BEGIN
	//================================================================================
	//SIEMENS AG // (c)Copyright 2019 All Rights Reserved
	//--------------------------------------------------------------------------------
	//Library:       LSimaHydTO
	//Tested with:   S7-15xx
	//Engineering:   TIA Portal  V15
	//Restrictions:  -
	//Requirements:  S7-1500 (FW 2.5)
	//Functionality: - for internal use
	//
	//--------------------------------------------------------------------------------
	//Change log table:
	//
	//Version     Date          Expert in charge    Changes applied
	//01.00.00    24.04.2020    APC_ERLF            First released version
	//================================================================================
	//
	
	#LSimaHydTO_GetSyncAxisCorrection := "LSimaHydTO_GetUnitsCorrection"(lengthUnit:=#axis.Units.LengthUnit,
	                                velocityUnit:=#axis.Units.VelocityUnit,
	                                accelFactor=>#accelFactor);
	
END_FUNCTION

FUNCTION_BLOCK "LSimaHydTO_HydraulicSimulationDrive"
{ S7_Optimized_Access := 'TRUE' }
AUTHOR : APC_ERLF
FAMILY : LSimaHydTO
VERSION : 1.22
   VAR_INPUT 
      enable : Bool;
      initPosition : LReal;
      minPosition : LReal := -1000000000000.0;
      maxPosition : LReal := 1000000000000.0;
      maxVelocity : LReal := 500.0;
      maxForce : LReal := 100.0;
      springDistance : LReal := 1.0;
      externalForce : LReal := 0.0;
      dynamicFrictionFactor : LReal;
      fixedStop : LReal := 1000000000000.0;
      fixedStopInverse : Bool;
      forceInverse : Bool;
      delayTime : LReal;
      cycleTime : UDInt;
      vChar_DB_NUMBER : UInt;
      axisTO : DB_ANY;
   END_VAR

   VAR_OUTPUT 
      busy { ExternalWritable := 'False'} : Bool;
      active { ExternalWritable := 'False'} : Bool;
      error { ExternalWritable := 'False'} : Bool;
      status { ExternalWritable := 'False'} : Word;
      simulatedPosition { ExternalWritable := 'False'} : LReal;
      simulatedForce { ExternalWritable := 'False'} : LReal;
      simulatedVChar { ExternalWritable := 'False'} : UInt;
      forceSensorAnalog_A { ExternalWritable := 'False'} : Word;
      forceSensorAnalog_B { ExternalWritable := 'False'} : Word;
   END_VAR

   VAR_IN_OUT 
      tel2in {InstructionName := 'PD_TEL2_IN'; LibVersion := '4.0'} : PD_TEL2_IN;
      tel2out {InstructionName := 'PD_TEL2_OUT'; LibVersion := '4.0'} : PD_TEL2_OUT;
      tel81in {InstructionName := 'PD_TEL81_IN'; LibVersion := '4.0'} : PD_TEL81_IN;
      tel81out {InstructionName := 'PD_TEL81_OUT'; LibVersion := '4.0'} : PD_TEL81_OUT;
   END_VAR

   VAR 
      statSetPoint { ExternalAccessible := 'False'; ExternalVisible := 'False'; ExternalWritable := 'False'} : LReal;
      statVelSetPoint { ExternalAccessible := 'False'; ExternalVisible := 'False'; ExternalWritable := 'False'} : LReal;
      statActualVChar { ExternalAccessible := 'False'; ExternalVisible := 'False'; ExternalWritable := 'False'} : UInt;
      statSampleTime { ExternalAccessible := 'False'; ExternalVisible := 'False'; ExternalWritable := 'False'} : LReal;
      statActualPosition { ExternalAccessible := 'False'; ExternalVisible := 'False'; ExternalWritable := 'False'} : LReal;
      statActualForce { ExternalAccessible := 'False'; ExternalVisible := 'False'; ExternalWritable := 'False'} : LReal;
      statForceFactor { ExternalAccessible := 'False'; ExternalVisible := 'False'; ExternalWritable := 'False'} : LReal;
      statEnableOld { ExternalAccessible := 'False'; ExternalVisible := 'False'; ExternalWritable := 'False'} : Bool;
      instSetPointPT1 { ExternalAccessible := 'False'; ExternalVisible := 'False'; ExternalWritable := 'False'} : "LSimaHydTO_T1";
      statPosLimitForce { ExternalAccessible := 'False'; ExternalVisible := 'False'; ExternalWritable := 'False'} : LReal;
      statNegLimitForce { ExternalAccessible := 'False'; ExternalVisible := 'False'; ExternalWritable := 'False'} : LReal;
      statFrictionForce { ExternalAccessible := 'False'; ExternalVisible := 'False'; ExternalWritable := 'False'} : LReal;
      instSimpleEncSetValue { ExternalAccessible := 'False'; ExternalVisible := 'False'; ExternalWritable := 'False'} : "LSimaHydTO_SimpleEncTel81";
      statVCharDB { ExternalAccessible := 'False'; ExternalVisible := 'False'; ExternalWritable := 'False'} : DB_ANY;
      statErrorVariant { ExternalAccessible := 'False'; ExternalVisible := 'False'; ExternalWritable := 'False'} : Int;
      instProfiDriveTel2 { ExternalAccessible := 'False'; ExternalVisible := 'False'; ExternalWritable := 'False'} : "LSimaHydTO_ProfiDriveTel2";
      statDriveEnabled { ExternalAccessible := 'False'; ExternalVisible := 'False'; ExternalWritable := 'False'} : Bool;
      statIntVelocityFactor { ExternalAccessible := 'False'; ExternalVisible := 'False'; ExternalWritable := 'False'} : LReal := 1.0;
   END_VAR

   VAR_TEMP 
      tempDeltaPosition : LReal;
      tempMinPos : LReal;
      tempMaxPos : LReal;
      tempActPosOld : LReal;
      tempVCharVar : Variant;
      tempRefToVChar : REF_TO "LSimaHydTO_typeVCharData";
      tempAccFactor : LReal;
   END_VAR

   VAR CONSTANT 
      ERR_INVALID_TYPE_OF_AXIS : Word := 16#8201;
   END_VAR


BEGIN
	//================================================================================
	//SIEMENS AG // (c)Copyright 2019 All Rights Reserved
	//--------------------------------------------------------------------------------
	//Library:       LSimaHydTO
	//Tested with:   S7-15xx
	//Engineering:   TIA Portal  V15
	//Restrictions:  -
	//Requirements:  S7-1500 (FW 2.5)
	//Functionality: Simulation of hydraulic axis   
	//
	//--------------------------------------------------------------------------------
	//Change log table:
	//
	//Version     Date          Expert in charge    Changes applied
	//01.00    15.03.2018    APC_ERLF            First released version
	//01.22    22.04.2020    APC_ERLF            improved: units are taken into account for the control
	//================================================================================
	
	
	IF #enable THEN
	  IF NOT #statEnableOld THEN //positive edge at enable
	    #error := FALSE;
	    #status := 16#0000;
	    #statSampleTime := UDINT_TO_LREAL(#cycleTime) * lreal#1.0E-9;
	    #statActualPosition := #initPosition;
	    
	    CASE TypeOfDB(#axisTO) OF
	            
	        TO_PositioningAxis:
	            #statIntVelocityFactor := "LSimaHydTO_GetPosAxisCorrection"(axis := #axisTO, accelFactor => #tempAccFactor);
	            
	        TO_SynchronousAxis:
	            #statIntVelocityFactor := "LSimaHydTO_GetSyncAxisCorrection"(axis := #axisTO, accelFactor => #tempAccFactor) ;
	            
	        ELSE
	            #error := TRUE;
	            #status := #ERR_INVALID_TYPE_OF_AXIS; // erorr
	            RETURN;
	    END_CASE;
	    
	    #busy := TRUE;
	    #active := TRUE;
	    
	    
	    
	  END_IF;
	  REGION evaluteVChar
	    IF #vChar_DB_NUMBER > 0 THEN
	      #statVCharDB := UINT_TO_DB_ANY(#vChar_DB_NUMBER);
	      #tempVCharVar := DB_ANY_TO_VARIANT(in := #statVCharDB, err => #statErrorVariant);
	      IF #statErrorVariant = 0 THEN
	        #tempRefToVChar ?= #tempVCharVar;
	        
	        IF TypeOf(#tempVCharVar) <> LSimaHydTO_typeVCharData THEN
	          #statErrorVariant := 8200;
	        END_IF;
	      END_IF;
	      IF #statErrorVariant <> 0 THEN
	        #statActualVChar := 0;
	        
	      ELSE
	        // check consinsesty of VChar
	        IF #tempRefToVChar^.MaxIdx < 1 OR #tempRefToVChar^.VelocityLimitPositive <= #tempRefToVChar^.VelocityLimitNegative THEN
	          #statActualVChar := 0;
	        ELSE
	          #statActualVChar := #vChar_DB_NUMBER;
	        END_IF;
	      END_IF;
	    ELSE
	      #statActualVChar := 0;
	    END_IF;
	    
	    #instProfiDriveTel2(setpoint => #statSetPoint,
	                        driveEnabled => #statDriveEnabled,
	                        tel2in := #tel2in,
	                        tel2out := #tel2out);
	    
	    
	    
	    IF #statActualVChar = 0 THEN
	      #statVelSetPoint := "LSimaHydTO_Scale"(input := #statSetPoint,
	                                           inBegin := -100.0,
	                                           inEnd := 100.0,
	                                           valBegin := - #maxVelocity,
	                                           valEnd := #maxVelocity);
	    ELSE
	      
	      #statVelSetPoint := "LSimaHydTO_VcharInverse"(qOutput := #statSetPoint, VChar := #tempRefToVChar^);
	      #statVelSetPoint := LIMIT(MN := - #maxVelocity, IN := #statVelSetPoint, MX := #maxVelocity);
	    END_IF;
	    #statVelSetPoint := #statVelSetPoint / #statIntVelocityFactor;
	    #simulatedVChar := #statActualVChar;
	  END_REGION
	  
	  #statActualForce := LIMIT(MN := - #maxForce, IN := #statActualForce, MX := #maxForce);
	  IF (#statActualForce > 0.0 AND
	    #statVelSetPoint > 0.0)
	    OR
	    (#statActualForce < 0.0 AND
	    #statVelSetPoint < 0.0)
	  THEN
	    #statForceFactor := MAX(IN1 := 0.0, IN2 := SQRT((#maxForce - ABS(#statActualForce)) / #maxForce));
	  ELSE
	    #statForceFactor := 1.0;
	  END_IF;
	  
	  
	  #instSetPointPT1(enable := #enable AND #delayTime > 0.0,
	                   inputValue := #statVelSetPoint,
	                   timeConstant := #delayTime,
	                   sampleTime := #statSampleTime
	                   // ,outputValue => 
	                   // ,active => 
	                   // ,error => 
	                   );
	  
	  #tempDeltaPosition := (#instSetPointPT1.outputValue) * #statSampleTime * #statForceFactor;
	  
	  //calculate AND LIMIT actual postition
	  #tempActPosOld := #statActualPosition;
	  
	  IF #fixedStopInverse THEN
	    #tempMinPos := LIMIT(MN := #minPosition
	                         , IN := #fixedStop
	                         , MX := #maxPosition);
	    #tempMaxPos := #maxPosition;
	  ELSE
	    #tempMinPos := #minPosition;
	    #tempMaxPos := LIMIT(MN := #minPosition
	                         , IN := #fixedStop
	                         , MX := #maxPosition);
	    
	  END_IF;
	  #statActualPosition := LIMIT( MN := #tempMinPos
	                              , IN := #tempActPosOld + #tempDeltaPosition
	                              , MX := #tempMaxPos
	                              );
	  #statFrictionForce := #dynamicFrictionFactor*(#statActualPosition - #tempActPosOld)/#statSampleTime;
	  IF #maxForce > 0.0
	    AND #springDistance > 0.0
	  THEN
	    
	    IF (#tempMaxPos - #statActualPosition) < #springDistance THEN
	      
	      #statPosLimitForce := LIMIT(MN := 0.0
	                                  , IN := (1 - (#tempMaxPos - #statActualPosition) / #springDistance) * #maxForce
	                                  , MX := #maxForce);
	    ELSE
	      #statPosLimitForce := 0.0;
	    END_IF;
	    IF (#statActualPosition - #tempMinPos) < #springDistance THEN
	      #statNegLimitForce := -LIMIT(MN := 0.0
	                                  , IN :=  (1 - (#statActualPosition - #tempMinPos) / #springDistance) * #maxForce
	                                  , MX := #maxForce);
	    ELSE
	      #statNegLimitForce := 0.0;
	    END_IF;
	    
	    #statActualForce := #externalForce + #statNegLimitForce + #statPosLimitForce + #statFrictionForce;
	    
	  ELSE
	    #statActualForce := #externalForce + #statFrictionForce;
	  END_IF;
	  
	  IF #forceInverse THEN
	    #statActualForce := -1.0 * #statActualForce;
	  END_IF;
	  //write actual position to technology object
	  
	  #simulatedPosition := #statActualPosition;
	  #simulatedForce := LIMIT(MN := - #maxForce, IN := #statActualForce, MX := #maxForce);
	  
	  IF #maxForce > 0.0 THEN
	    IF #simulatedForce >= 0.0 THEN
	      #forceSensorAnalog_A := INT_TO_WORD(LREAL_TO_INT(#simulatedForce * 27648.0 / #maxForce));
	      #forceSensorAnalog_B := 0;
	    ELSE
	      #forceSensorAnalog_B := INT_TO_WORD(LREAL_TO_INT(ABS(#simulatedForce) * 27648.0 / #maxForce));
	      #forceSensorAnalog_A := 0;
	    END_IF;
	  ELSE
	    #forceSensorAnalog_A := 0;
	    #forceSensorAnalog_B := 0;
	  END_IF;
	  
	  #instSimpleEncSetValue(position := #simulatedPosition,
	                         init := #enable AND NOT #statEnableOld,
	                         axis:=#axisTO,
	                         status=>#status,
	                         tel81in := #tel81in,
	                         tel81out := #tel81out);
	  
	  
	  
	ELSE
	  IF #statEnableOld THEN //negative edge
	    #busy := FALSE;
	    #active := FALSE;
	    #simulatedVChar := 0;
	    
	    #statActualPosition := 0.0;
	    #statActualForce := 0.0;
	    #simulatedPosition := 0.0;
	    #simulatedForce := 0.0;
	    #forceSensorAnalog_A := 0;
	    #forceSensorAnalog_B := 0;
	  END_IF;
	END_IF;
	
	
	#statEnableOld := #enable;
	
	
	
	
	
	
END_FUNCTION_BLOCK

FUNCTION_BLOCK "LSimaHydTO_ProfiDriveTel2"
{ S7_Optimized_Access := 'FALSE' }
AUTHOR : APC_ERLF
FAMILY : LSimaHydTO
VERSION : 1.0
   VAR_OUTPUT 
      setpoint { ExternalAccessible := 'False'; ExternalVisible := 'False'; ExternalWritable := 'False'} : LReal;
      driveEnabled { ExternalAccessible := 'False'; ExternalVisible := 'False'; ExternalWritable := 'False'} : Bool;
   END_VAR

   VAR_IN_OUT 
      tel2in {InstructionName := 'PD_TEL2_IN'; LibVersion := '4.0'} : PD_TEL2_IN;
      tel2out {InstructionName := 'PD_TEL2_OUT'; LibVersion := '4.0'} : PD_TEL2_OUT;
   END_VAR

   VAR 
      statZSW1 {InstructionName := 'PD_ZSW1'; LibVersion := '4.0'; ExternalAccessible := 'False'; ExternalVisible := 'False'; ExternalWritable := 'False'} : PD_ZSW1;
      statWZSW1 { ExternalAccessible := 'False'; ExternalVisible := 'False'; ExternalWritable := 'False'} AT statZSW1 : Word;
   END_VAR

   VAR_TEMP 
      tempNsollSigned : DInt;
   END_VAR

   VAR CONSTANT 
      ZSW1_S1 : Word := 2#0000_0011_0111_0000;
      ZSW1_S2 : Word := 2#0000_0011_0011_0001;
      ZSW1_S3 : Word := 2#0000_0011_0011_0011;
      ZSW1_S4 : Word := 2#0000_0011_0011_0111;
      C_100_PROZENT : LReal := 10737418.24;
   END_VAR


BEGIN
	//================================================================================
	//SIEMENS AG // (c)Copyright 2019 All Rights Reserved
	//--------------------------------------------------------------------------------
	//Library:       LSimaHydTO
	//Tested with:   S7-15xx
	//Engineering:   TIA Portal  V15
	//Restrictions:  -
	//Requirements:  S7-1500 (FW 2.5)
	//Functionality: Support of drive transmitter   
	//
	//--------------------------------------------------------------------------------
	//Change log table:
	//
	//Version     Date          Expert in charge    Changes applied
	//01.00.00    29.03.2017    APC_ERLF            First released version
	//================================================================================
	
	
	IF #tel2out.STW1.NoCoastStop AND #tel2out.STW1.NoQuickStop THEN
	    IF #tel2out.STW1.On THEN
	        IF #tel2out.STW1.EnableOperation THEN
	            #statWZSW1 := #ZSW1_S4;             // operation
	            #driveEnabled := TRUE;
	        ELSE
	            #statWZSW1 := #ZSW1_S3;             // switched on
	        END_IF;
	    ELSE
	        #statWZSW1 := #ZSW1_S2;                 // ready for switch on
	    END_IF;
	ELSE
	    #statWZSW1 := #ZSW1_S1;                 // coast stop, quick stop
	    #driveEnabled := FALSE;
	END_IF;
	#tel2in.ZSW1 := #statZSW1;
	//-----------------  Interface -----------  
	#tempNsollSigned := DWORD_TO_DINT(#tel2out.NSOLL_B); // NSOLL is really a signed DINT
	#setpoint := DINT_TO_LREAL(#tempNsollSigned)/#C_100_PROZENT;      // desired speed 
	IF #statWZSW1 = #ZSW1_S4 THEN
	  #tel2in.NIST_B := #tel2out.NSOLL_B;
	ELSE
	  #tel2in.NIST_B := 0;
	END_IF;
	
	
END_FUNCTION_BLOCK

FUNCTION "Scale" : Void   // FC1, LAD
{ S7_Optimized_Access := 'TRUE' }
VERSION : 0.1
// stored: AutoNumber true, IsIECCheckEnabled false, SetENOAutomatically false, UDAEnableTagReadback false
   VAR_OUTPUT
      Scale_Out : Real;
   END_VAR
   VAR_TEMP
      AUX : Real;
   END_VAR
BEGIN

REGION Network 1
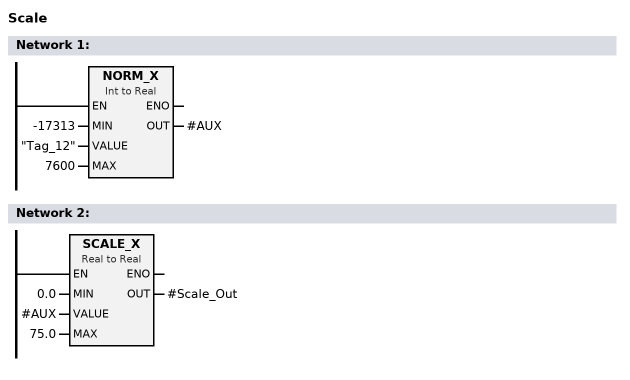
   RUNG wire#powerrail
      { S7_Templates := "[SrcType := Int, DestType := Real]" } Normalize(min := -17313, value := "Tag_12", max := 7600, out => #AUX)
   END_RUNG
   // the same network as SCL:
   #AUX := NORM_X(MIN := -17313, VALUE := "Tag_12", MAX := 7600);
END_REGION

REGION Network 2
   RUNG wire#powerrail
      { S7_Templates := "[SrcType := Real, DestType := Real]" } Scale(min := 0.0, value := #AUX, max := 75.0, out => #Scale_Out)
   END_RUNG
   // the same network as SCL:
   #Scale_Out := SCALE_X(MIN := 0.0, VALUE := #AUX, MAX := 75.0);
END_REGION
END_FUNCTION

ORGANIZATION_BLOCK "SimaHydTO_Main_HMI"   // OB124, LAD, ProgramCycle
TITLE = SimaHydTO_Main_HMI
{ S7_Optimized_Access := 'TRUE' }
FAMILY : SimaHydTO
VERSION : 1.0
// Organization block information: See Organization block network 1
// stored: AutoNumber true, IsIECCheckEnabled false, SetENOAutomatically false
   VAR_INPUT
      Initial_Call : Bool;   // Initial call of this OB
      Remanence : Bool;   // =True, if remanent data are available
   END_VAR
BEGIN

REGION Network 1 (SCL): SimaHydTO - HMI Interface
   //=============================================================================
   //SIEMENS AG
   //(c)Copyright 2016 All Rights Reserved
   //-----------------------------------------------------------------------------
   //Library:       OB of LSimaHydTO_HMI
   //Tested with:   S7-1500 V2.5
   //Engineering:   TIA Portal V15
   //Restrictions:  -
   //Requirements:  S7-1500(T)
   //Functionality: Connection between HMI and PLC program
   //-----------------------------------------------------------------------------
   //Change log table:
   //Version  Date       Expert in charge Changes applied
   //01.00.00 18.07.2019 ArSc             First released version
   //=============================================================================
END_REGION

REGION Network 2: SimaHydTO - HMI Interface: Function calls of HMI functionality
   // Controlling the functionality of SimaHydTO via HMI
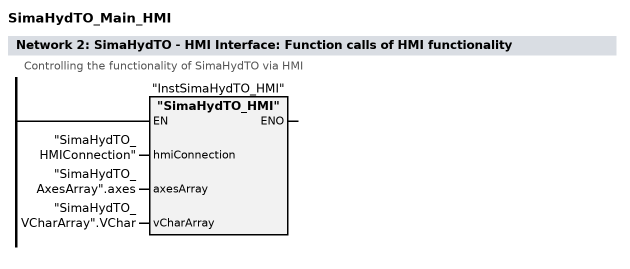
   RUNG wire#powerrail
      "InstSimaHydTO_HMI"(hmiConnection := "SimaHydTO_HMIConnection", axesArray := "SimaHydTO_AxesArray".axes, vCharArray := "SimaHydTO_VCharArray".VChar)
   END_RUNG
   // the same network as SCL:
   "InstSimaHydTO_HMI"(hmiConnection := "SimaHydTO_HMIConnection",   // "SimaHydTO_HMI"
                       axesArray := "SimaHydTO_AxesArray".axes,
                       vCharArray := "SimaHydTO_VCharArray".VChar);
END_REGION
END_ORGANIZATION_BLOCK

FUNCTION_BLOCK "SimaHydTO_HMI"
{ S7_Optimized_Access := 'TRUE' }
FAMILY : SimaHydTO
VERSION : 1.0
   VAR_IN_OUT 
      hmiConnection : "SimaHydTO_typeHMIConnection";
      axesArray : Array[*] of "SimaHydTO_typeAxesArray";
      vCharArray : Array[*] of "SimaHydTO_typeVCharArray";
   END_VAR

   VAR 
      statInitObjects { ExternalAccessible := 'False'; ExternalVisible := 'False'; ExternalWritable := 'False'} : Bool := TRUE;
      instHmiAxisSelector { ExternalAccessible := 'False'; ExternalVisible := 'False'; ExternalWritable := 'False'} : "SimaHydTO_HmiAxisSelector";
      instHmiVCharSelector { ExternalAccessible := 'False'; ExternalVisible := 'False'; ExternalWritable := 'False'} : "SimaHydTO_HmiVCharSelector";
      instBasicAxisControl { ExternalAccessible := 'False'; ExternalVisible := 'False'; ExternalWritable := 'False'} : "SimaHydTO_BasicAxisControl";
      instVCharMeasurement { ExternalAccessible := 'False'; ExternalVisible := 'False'; ExternalWritable := 'False'} : "SimaHydTO_VCharMeasurement";
      instVCharEditor { ExternalAccessible := 'False'; ExternalVisible := 'False'; ExternalWritable := 'False'} : "SimaHydTO_VCharEditor";
      instAdvancedAxisControl { ExternalAccessible := 'False'; ExternalVisible := 'False'; ExternalWritable := 'False'} : "SimaHydTO_AdvancedAxisControl";
      instParameterSettings { ExternalAccessible := 'False'; ExternalVisible := 'False'; ExternalWritable := 'False'} : "SimaHydTO_ParameterSettings";
      instFindVChars { ExternalAccessible := 'False'; ExternalVisible := 'False'; ExternalWritable := 'False'} : "SimaHydTO_FindObjects";
      instVCharManagement { ExternalAccessible := 'False'; ExternalVisible := 'False'; ExternalWritable := 'False'} : "SimaHydTO_VCharManagement";
   END_VAR

   VAR_TEMP 
      tempVariant : Variant;
      tempErrorVariant : Int;
      tempDbAny : DB_ANY;
      tempHydAxisData : REF_TO "LSimaHydTO_typeAxisData";
   END_VAR


BEGIN
	//=============================================================================
	//SIEMENS AG
	//(c)Copyright 2016 All Rights Reserved
	//-----------------------------------------------------------------------------
	//Library:       SimaHydTO_HMI
	//Tested with:   S7-1500 V2.5
	//Engineering:   TIA Portal V15
	//Restrictions:  -
	//Requirements:  S7-1500(T)
	//Functionality: Connection between HMI and PLC program
	//-----------------------------------------------------------------------------
	//Change log table:
	//Version  Date       Expert in charge Changes applied
	//01.00.00 12.07.2019 ArSc             First released version
	//=============================================================================
	
	#instFindVChars(execute := #statInitObjects,
	                axesArray := #axesArray,
	                vCharArray := #vCharArray);
	IF NOT #instFindVChars.busy THEN
	  #statInitObjects := FALSE;
	END_IF;
	
	//=============================================================================
	//Axis selector
	//=============================================================================
	
	//Axis selection 
	#instHmiAxisSelector(selector := #hmiConnection.AxisSelector,
	                     axesArray := #axesArray);
	
	
	
	//===================================================================================
	//evalute objects
	//
	
	#tempDbAny := #hmiConnection.AxisSelector.Status.selectedAxis;
	#tempVariant := DB_ANY_TO_VARIANT(in := #tempDbAny, err => #tempErrorVariant);
	
	IF TypeOf(#tempVariant) = LSimaHydTO_typeAxisData THEN
	  #tempHydAxisData ?= #tempVariant;
	  
	END_IF;
	//=============================================================================
	//Basic axis control
	//=============================================================================
	
	//Check axis selection
	IF (#hmiConnection.AxisSelector.Status.dataValid = True)
	THEN
	  IF (#hmiConnection.AxisSelector.Status.selectionChanged = True)
	  THEN
	    CASE #hmiConnection.AxisSelector.Status.selectedTypeOfAxis OF
	      2: //posaxis
	        #hmiConnection.AxisToData.axisUnits := "SimaHydTO_GetAxisToUnits_PosAxis"(#hmiConnection.AxisSelector.Status.selectedTO_Axis);
	        
	      3: // syncaxis
	        #hmiConnection.AxisToData.axisUnits := "SimaHydTO_GetAxisToUnits_SyncAxis"(#hmiConnection.AxisSelector.Status.selectedTO_Axis);
	        
	    END_CASE;
	    #hmiConnection.AxisToData.typeOfAxis := #hmiConnection.AxisSelector.Status.selectedTypeOfAxis;
	  END_IF;
	  
	  // Axis animation
	    "SimaHydTO_HmiAxisAnimation"(hmiConnection := #hmiConnection,
	                                 axisData := #tempHydAxisData^);
	    
	  
	  
	  //Transfer data between axis and HMI
	  #instBasicAxisControl(hmiConnection := #hmiConnection,
	                        axisData := #tempHydAxisData^,
	                        axesArray := #axesArray);
	  
	  
	  
	  //=============================================================================
	  //VChar measurement
	  //=============================================================================
	  
	  //Call function block
	  #instVCharMeasurement(hmiConnection := #hmiConnection,
	                        axisData := #tempHydAxisData^,
	                        axesArray:=#axesArray,
	                        vCharArray := #vCharArray);
	  
	  
	  
	  //=============================================================================
	  //Advanced axis control
	  //=============================================================================
	  #instAdvancedAxisControl(hmiConnection := #hmiConnection,
	                           axisData := #tempHydAxisData^,
	                           axesArray := #axesArray);
	  
	  
	  #instVCharManagement(hmiConnection:=#hmiConnection,
	                       axisData:=#tempHydAxisData^,
	                       vCharArray:=#vCharArray);
	
	  
	ELSE
	  //In case of no valid data of axis selection, do nothing...
	  ;
	END_IF;
	
	//=============================================================================
	//VChar editor
	//=============================================================================
	
	//Do function...
	#instVCharEditor(hmiConnection := #hmiConnection,
	                 vCharArray := #vCharArray);
	
	
	
	//=============================================================================
	//Parameter settings
	//=============================================================================
	
	//Check axis selection
	//Do function...
	#instParameterSettings(hmiConnection := #hmiConnection,
	                       axisData := #tempHydAxisData^,
	                       VCharArray := #vCharArray);
	
	
	
	
	
END_FUNCTION_BLOCK

FUNCTION_BLOCK "SimaHydTO_HmiAxisSelector"
{ S7_Optimized_Access := 'TRUE' }
FAMILY : SimaHydTO
VERSION : 1.0
   VAR_IN_OUT 
      selector : "SimaHydTO_typeHMIConnectionAxisSelector";
      axesArray : Array[*] of "SimaHydTO_typeAxesArray";
   END_VAR

   VAR 
      statFirstRunDone { ExternalAccessible := 'False'; ExternalVisible := 'False'; ExternalWritable := 'False'} : Bool;
      statActualAxisIndex { ExternalAccessible := 'False'; ExternalVisible := 'False'; ExternalWritable := 'False'} : Int;
      statArrayMinIndex { ExternalAccessible := 'False'; ExternalVisible := 'False'; ExternalWritable := 'False'} : Int;
      statArrayMaxIndex { ExternalAccessible := 'False'; ExternalVisible := 'False'; ExternalWritable := 'False'} : Int;
      statPreviousObjectOld { ExternalAccessible := 'False'; ExternalVisible := 'False'; ExternalWritable := 'False'} : Bool;
      statNextObjectOld { ExternalAccessible := 'False'; ExternalVisible := 'False'; ExternalWritable := 'False'} : Bool;
      statExecuteDirectIndexSelectionOld { ExternalAccessible := 'False'; ExternalVisible := 'False'; ExternalWritable := 'False'} : Bool;
      statActualAxisIndexOld { ExternalAccessible := 'False'; ExternalVisible := 'False'; ExternalWritable := 'False'} : Int;
   END_VAR

   VAR_TEMP 
      tempVariant : Variant;
      tempErrorVariant : Int;
      tempDbAny : DB_ANY;
      tempHydAxisData : REF_TO "LSimaHydTO_typeAxisData";
   END_VAR

   VAR CONSTANT 
      ERROR_AXIS_INDEX : Int := 0;
      ERROR_SELECTED_HYDAXIS : DB_ANY := 0;
      ERROR_SELECTED_HYDAXIS_INTEGER : UInt := 0;
      ERROR_SELECTED_HYDAXIS_NAME : WString := WSTRING#'';
      ERROR_SELECTED_AXISTO : DB_ANY := 0;
      ERROR_SELECTED_AXISTO_INTEGER : UInt := 0;
      ERROR_SELECTED_AXISTO_TYPE : Int := 0;
      ERROR_SELECTED_VCHAR : DB_ANY := 0;
      ERROR_SELECTED_VCHAR_INTEGER : UInt := 0;
   END_VAR


BEGIN
	//=============================================================================
	//SIEMENS AG
	//(c)Copyright 2016 All Rights Reserved
	//-----------------------------------------------------------------------------
	//Library:       SimaHydTO_HMI
	//Tested with:   S7-1500 V2.5
	//Engineering:   TIA Portal V15
	//Restrictions:  -
	//Requirements:  S7-1500(T)
	//Functionality: Selection of hydraulic axis out of axis array
	//-----------------------------------------------------------------------------
	//Change log table:
	//Version  Date       Expert in charge Changes applied
	//01.00.00 12.07.2019 ArSc             First released version
	//=============================================================================
	
	
	//Array detection and initialization
	IF (#statFirstRunDone = False)
	THEN
	  //Get MIN and MAX of array indices
	  #statArrayMinIndex := DINT_TO_INT(LOWER_BOUND(ARR := #axesArray, DIM := 1));
	  #statArrayMaxIndex := DINT_TO_INT(UPPER_BOUND(ARR := #axesArray, DIM := 1));
	  //Set default value of actual axis index
	  #statActualAxisIndex := #statArrayMinIndex;
	  #statActualAxisIndexOld := #statArrayMinIndex-1;
	  //Mark first run of function block
	  #statFirstRunDone := True;
	  #selector.Status.dataError := False;
	  #selector.Status.dataValid := False;
	END_IF;
	  //Select axis (in axis data array)
	  //Previous axis
	IF ((#selector.Command.previousObject = True)
	    AND (#statPreviousObjectOld = False)
	    AND (#selector.Command.nextObject = False)
	    AND (#selector.Command.executeDirectIndexSelection = False))
	  THEN
	    //Decrement actual axis index
	    #statActualAxisIndex := #statActualAxisIndex - INT#1;
	    //Check index minimum
	    IF (#statActualAxisIndex < #statArrayMinIndex)
	    THEN
	      //Select last axis by index
	      #statActualAxisIndex := #statArrayMaxIndex;
	    END_IF;
	    //Next axis  
	  ELSIF ((#selector.Command.nextObject = True)
	    AND (#statNextObjectOld = False)
	    AND (#selector.Command.previousObject = False)
	    AND (#selector.Command.executeDirectIndexSelection = False))
	  THEN
	    //Increment actual axis index
	    #statActualAxisIndex := #statActualAxisIndex + INT#1;
	    //Check index minimum
	    IF (#statActualAxisIndex > #statArrayMaxIndex)
	    THEN
	      //Select first axis by index
	      #statActualAxisIndex := #statArrayMinIndex;
	    END_IF;
	    //Direct selection
	  ELSIF ((#selector.Command.executeDirectIndexSelection = True)
	    AND (#statExecuteDirectIndexSelectionOld = False)
	    AND (#selector.Command.nextObject = False)
	    AND (#selector.Command.previousObject = False))
	  THEN
	    IF ((#selector.Command.directIndexSelection >= #statArrayMinIndex)
	      AND (#selector.Command.directIndexSelection <= #statArrayMaxIndex))
	    THEN
	      //Set axis index directly
	      #statActualAxisIndex := #selector.Command.directIndexSelection;
	    END_IF;
	  END_IF;
	
	  #selector.Status.selectionChanged := FALSE;
	  IF #statActualAxisIndex <> #statActualAxisIndexOld
	    AND #axesArray[#statActualAxisIndex].initialized
	  THEN
	    //Write function block output
	    #selector.Status.actualAxisIndex := #statActualAxisIndex;
	    #tempDbAny := #axesArray[#statActualAxisIndex].axisData;
	    
	    #selector.Status.selectedAxis := #tempDbAny;
	    #selector.Status.selectedAxisInteger := DB_ANY_TO_UINT(#tempDbAny);
	    
	    //Get axis data
	    #tempVariant := DB_ANY_TO_VARIANT(in := #tempDbAny, err => #tempErrorVariant);
	    
	    IF TypeOf(#tempVariant) = LSimaHydTO_typeAxisData THEN
	      #tempHydAxisData ?= #tempVariant;
	      
	      //Read hydraulic axis name
	      #selector.Status.selectedAxisName := #tempHydAxisData^.Name;
	      //Read connected technology object axis
	      
	      CASE TypeOfDB(#tempHydAxisData^.TO_Axis) OF
	          
	        TO_PositioningAxis:
	          #selector.Status.selectedTO_Axis := #tempHydAxisData^.TO_Axis;
	          #selector.Status.selectedAxisTOInteger := DB_ANY_TO_UINT(#selector.Status.selectedTO_Axis);
	          #selector.Status.selectedTypeOfAxis := 2;
	          
	          #selector.Status.dataValid := TRUE;
	          
	        TO_SynchronousAxis:
	          #selector.Status.selectedTO_Axis := #tempHydAxisData^.TO_Axis;
	          #selector.Status.selectedAxisTOInteger := DB_ANY_TO_UINT(#selector.Status.selectedTO_Axis);
	          #selector.Status.selectedTypeOfAxis := 3;
	          #selector.Status.dataValid := TRUE;
	          
	        ELSE
	          #selector.Status.selectedTO_Axis := 0;
	          #selector.Status.selectedAxisTOInteger := 0;
	          #selector.Status.selectedTypeOfAxis := 0;
	          #selector.Status.dataValid := FALSE;
	          
	      END_CASE;
	      //Read active valve characteristics
	      #selector.Status.selectedVChar := #tempHydAxisData^.ValveCharacteristic.DB_NUMBER;
	      #selector.Status.selectedVCharInteger := DB_ANY_TO_UINT(#selector.Status.selectedVChar);
	      
	      //Write function block output
	      #selector.Status.dataError := False;
	  //    #selector.Status.dataValid := TRUE;
	      #selector.Status.selectionChanged := TRUE;
	    ELSE
	      //error handling
	      #selector.Status.dataError := True;
	      #selector.Status.dataValid := False;
	      
	      #selector.Status.actualAxisIndex := #statActualAxisIndex;
	      #selector.Status.selectedAxis := #ERROR_SELECTED_HYDAXIS;
	      #selector.Status.selectedAxisInteger := #ERROR_SELECTED_HYDAXIS_INTEGER;
	      #selector.Status.selectedAxisName := #ERROR_SELECTED_HYDAXIS_NAME;
	      #selector.Status.selectedTO_Axis := #ERROR_SELECTED_AXISTO;
	      #selector.Status.selectedAxisTOInteger := #ERROR_SELECTED_AXISTO_INTEGER;
	      #selector.Status.selectedTypeOfAxis := #ERROR_SELECTED_AXISTO_TYPE;
	      #selector.Status.selectedVChar := #ERROR_SELECTED_VCHAR;
	      #selector.Status.selectedVCharInteger := #ERROR_SELECTED_VCHAR_INTEGER;
	      
	    END_IF;
	    //Save AxisIndex for edge control
	    #statActualAxisIndexOld := #statActualAxisIndex;
	    
	  END_IF;
	
	
	//-----------------------------------------------------------------------------
	//Function block system functions
	//-----------------------------------------------------------------------------
	
	//Save signals for edge control
	  #statPreviousObjectOld := #selector.Command.previousObject;
	  #statNextObjectOld := #selector.Command.nextObject;
	  #statExecuteDirectIndexSelectionOld := #selector.Command.executeDirectIndexSelection;
	
	
	
END_FUNCTION_BLOCK

FUNCTION_BLOCK "SimaHydTO_HmiVCharSelector"
{ S7_Optimized_Access := 'TRUE' }
FAMILY : SimaHydTO
VERSION : 1.0
   VAR_INPUT 
      command { ExternalAccessible := 'False'; ExternalVisible := 'False'; ExternalWritable := 'False'} : "SimaHydTO_typeHMIConnectionVCharSelectorCommand";
   END_VAR

   VAR_IN_OUT 
      status : "SimaHydTO_typeHMIConnectionVCharSelectorStatus";
      vCharArray : Array[*] of "SimaHydTO_typeVCharArray";
   END_VAR

   VAR 
      statFirstRunDone { ExternalAccessible := 'False'; ExternalVisible := 'False'; ExternalWritable := 'False'} : Bool;
      statActualVCharIndex { ExternalAccessible := 'False'; ExternalVisible := 'False'; ExternalWritable := 'False'} : Int;
      statArrayMinIndex { ExternalAccessible := 'False'; ExternalVisible := 'False'; ExternalWritable := 'False'} : Int;
      statArrayMaxIndex { ExternalAccessible := 'False'; ExternalVisible := 'False'; ExternalWritable := 'False'} : Int;
      statPreviousObjectOld { ExternalAccessible := 'False'; ExternalVisible := 'False'; ExternalWritable := 'False'} : Bool;
      statNextObjectOld { ExternalAccessible := 'False'; ExternalVisible := 'False'; ExternalWritable := 'False'} : Bool;
      statExecuteDirectIndexSelectionOld { ExternalAccessible := 'False'; ExternalVisible := 'False'; ExternalWritable := 'False'} : Bool;
   END_VAR

   VAR_TEMP 
      tempVariant : Variant;
      tempErrorVariant : Int;
      tempDbAny : DB_ANY;
      tempVCharData : REF_TO "LSimaHydTO_typeVCharData";
      tempIndexChanged : Bool;
   END_VAR

   VAR CONSTANT 
      ERROR_VCHAR_INDEX : Int := 0;
      ERROR_SELECTED_VCHAR : DB_ANY := 0;
      ERROR_SELECTED_VCHAR_INTEGER : UInt := 0;
      ERROR_SELECTED_VCHAR_NAME : WString := WSTRING#'';
   END_VAR


BEGIN
	//=============================================================================
	//SIEMENS AG
	//(c)Copyright 2016 All Rights Reserved
	//-----------------------------------------------------------------------------
	//Library:       SimaHydTO_HMI
	//Tested with:   S7-1500 V2.5
	//Engineering:   TIA Portal V15
	//Restrictions:  -
	//Requirements:  S7-1500(T)
	//Functionality: Selection of VChar (valve characteristics) controlled via HMI
	//-----------------------------------------------------------------------------
	//Change log table:
	//Version  Date       Expert in charge Changes applied
	//01.00.00 12.07.2019 ArSc             First released version
	//=============================================================================
	
	
	//Array detection and initialization
	IF (#statFirstRunDone = False)
	THEN
	  //Get MIN and MAX of array indices
	  #statArrayMinIndex := DINT_TO_INT(LOWER_BOUND(ARR := #vCharArray, DIM := 1));
	  #statArrayMaxIndex := DINT_TO_INT(UPPER_BOUND(ARR := #vCharArray, DIM := 1));
	  //Set default value of actual axis index
	  #statActualVCharIndex := #statArrayMinIndex;
	  //Mark first run of function block
	  IF #vCharArray[#statActualVCharIndex].initialized THEN
	    #statFirstRunDone := True;
	    #tempIndexChanged := TRUE;
	  END_IF;
	  
	ELSE
	  //Select axis (in axis data array)
	  //Previous axis
	  IF (#command.previousObject
	    AND  NOT #statPreviousObjectOld)
	  THEN
	    //Decrement actual axis index
	    #statActualVCharIndex := #statActualVCharIndex - INT#1;
	    //Check index minimum
	    IF (#statActualVCharIndex < #statArrayMinIndex)
	    THEN
	      //Select last axis by index
	      #statActualVCharIndex := #statArrayMaxIndex;
	    END_IF;
	    #tempIndexChanged := TRUE;
	  //Next axis  
	  ELSIF (#command.nextObject
	    AND NOT #statNextObjectOld)
	  THEN
	    //Increment actual axis index
	    #statActualVCharIndex := #statActualVCharIndex + INT#1;
	    //Check index minimum
	    IF (#statActualVCharIndex > #statArrayMaxIndex)
	    THEN
	      //Select first axis by index
	      #statActualVCharIndex := #statArrayMinIndex;
	    END_IF;
	    #tempIndexChanged := TRUE;
	  //Direct selection
	  ELSIF (#command.executeDirectIndexSelection
	    AND NOT #statExecuteDirectIndexSelectionOld)
	  THEN
	    IF ((#command.directIndexSelection >= #statArrayMinIndex)
	      AND (#command.directIndexSelection <= #statArrayMaxIndex))
	    THEN
	      //Set axis index directly
	      #statActualVCharIndex := DINT_TO_INT(#command.directIndexSelection);
	      #tempIndexChanged := TRUE;
	    END_IF;
	  END_IF;
	END_IF;
	
	
	IF (#statFirstRunDone)
	THEN
	  //Write function block output
	  #status.actualVCharIndex := #statActualVCharIndex;
	  IF #tempIndexChanged  THEN
	    //Get VChar data
	    #tempDbAny := #vCharArray[#status.actualVCharIndex].VChar_DB;
	    #tempVariant := DB_ANY_TO_VARIANT(in := #tempDbAny, err => #tempErrorVariant);
	    
	    IF TypeOf(#tempVariant) = LSimaHydTO_typeVCharData THEN
	      #tempVCharData ?= #tempVariant;
	      
	      #status.selectedVChar := #vCharArray[#status.actualVCharIndex].VChar_DB;
	      #status.selectedVCharName := #tempVCharData^.Name;
	      #status.selectedVCharInteger := DB_ANY_TO_UINT(#status.selectedVChar);
	      
	      //Write function block output
	      #status.dataError := False;
	      #status.dataValid := True;
	      
	    ELSE
	      //error handling
	      #status.dataError := True;
	      #status.dataValid := False;
	      
	      // #actualVCharIndex := #ERROR_VCHAR_INDEX;
	      #status.selectedVChar := #ERROR_SELECTED_VCHAR;
	      #status.selectedVCharInteger := #ERROR_SELECTED_VCHAR_INTEGER;
	      #status.selectedVCharName := #ERROR_SELECTED_VCHAR_NAME;
	      
	    END_IF;
	    #tempIndexChanged := FALSE;
	  END_IF;
	ELSE
	  //Write function block output
	  #status.dataError := False;
	  #status.dataValid := False;
	END_IF;
	
	
	//-----------------------------------------------------------------------------
	//Function block system functions
	//-----------------------------------------------------------------------------
	
	//Save signals for edge control
	#statPreviousObjectOld := #command.previousObject;
	#statNextObjectOld := #command.nextObject;
	#statExecuteDirectIndexSelectionOld := #command.executeDirectIndexSelection;
	//Save AxisIndex for edge control
	
	
	
END_FUNCTION_BLOCK

FUNCTION_BLOCK "SimaHydTO_BasicAxisControl"
{ S7_Optimized_Access := 'TRUE' }
FAMILY : SimaHydTO
VERSION : 1.0
   VAR_IN_OUT 
      hmiConnection : "SimaHydTO_typeHMIConnection";
      axisData : "LSimaHydTO_typeAxisData";
      axesArray : Array[*] of "SimaHydTO_typeAxesArray";
   END_VAR

   VAR 
      statActualAxisIndex { ExternalAccessible := 'False'; ExternalVisible := 'False'; ExternalWritable := 'False'} : Int;
      statAxisIndexOld { ExternalAccessible := 'False'; ExternalVisible := 'False'; ExternalWritable := 'False'} : Int := -1;
      instAxisBasicsPosAxis { ExternalAccessible := 'False'; ExternalVisible := 'False'; ExternalWritable := 'False'} : "SimaHydTO_AxisBasics_PosAxis";
      instAxisBasicsSyncAxis { ExternalAccessible := 'False'; ExternalVisible := 'False'; ExternalWritable := 'False'} : "SimaHydTO_AxisBasics_SyncAxis";
      instDirectOutputControl { ExternalAccessible := 'False'; ExternalVisible := 'False'; ExternalWritable := 'False'} : "LSimaHydTO_MC_DirectOutputControl";
      instLSimaHydTO_MC_RequestDirection { ExternalAccessible := 'False'; ExternalVisible := 'False'; ExternalWritable := 'False'} : "LSimaHydTO_MC_RequestDirection";
      instLSimaHydTO_MC_Reset { ExternalAccessible := 'False'; ExternalVisible := 'False'; ExternalWritable := 'False'} : "LSimaHydTO_MC_Reset";
   END_VAR


BEGIN
	//=============================================================================
	//SIEMENS AG
	//(c)Copyright 2016 All Rights Reserved
	//-----------------------------------------------------------------------------
	//Library:       SimaHydTO_BasicAxisControl
	//Tested with:   S7-1500 V2.5
	//Engineering:   TIA Portal V15
	//Restrictions:  -
	//Requirements:  S7-1500(T)
	//Functionality: Transfer data from/to HMI to/from selected axis
	//-----------------------------------------------------------------------------
	//Change log table:
	//Version  Date       Expert in charge Changes applied
	//01.00.00 12.07.2019 ArSc             First released version
	//=============================================================================
	
	
	//Check axis selection, if axis has changed
	IF  #hmiConnection.AxisSelector.Status.selectionChanged
	  AND #hmiConnection.AxisSelector.Status.dataValid
	THEN
	  //Preset axis commands
	  #statActualAxisIndex := #hmiConnection.AxisSelector.Status.actualAxisIndex;
	  IF #statAxisIndexOld > -1 THEN
	    //Save axis commands
	    #axesArray[#statAxisIndexOld].basicControl := #hmiConnection.BasicAxisControl.Command;
	    #axesArray[#statAxisIndexOld].basicControl.homeExecute := FALSE;
	    #axesArray[#statAxisIndexOld].basicControl.jogBackward := FALSE;
	    #axesArray[#statAxisIndexOld].basicControl.jogForward := FALSE;
	    #axesArray[#statAxisIndexOld].basicControl.resetExecute := FALSE;
	    #axesArray[#statAxisIndexOld].basicControl.resetFBExecute := FALSE;
	    
	    #axesArray[#statAxisIndexOld].directOutputControl := #hmiConnection.BasicAxisControl.ControlDirectOutput;
	    #axesArray[#statAxisIndexOld].directOutputControl.jogForward := FALSE;
	    #axesArray[#statAxisIndexOld].directOutputControl.jogBackward := FALSE;
	  END_IF;
	  
	  
	  #hmiConnection.BasicAxisControl.Command := #axesArray[#statActualAxisIndex].basicControl;
	  #hmiConnection.BasicAxisControl.Command.homeExecute := FALSE;
	  #hmiConnection.BasicAxisControl.Command.jogBackward := FALSE;
	  #hmiConnection.BasicAxisControl.Command.jogForward := FALSE;
	  #hmiConnection.BasicAxisControl.Command.resetExecute := FALSE;
	  #hmiConnection.BasicAxisControl.Command.resetFBExecute := FALSE;
	  //Preset manual output paramter and commands
	  #hmiConnection.BasicAxisControl.ControlDirectOutput := #axesArray[#statActualAxisIndex].directOutputControl;
	  #hmiConnection.BasicAxisControl.ControlDirectOutput.jogBackward := FALSE;
	  #hmiConnection.BasicAxisControl.ControlDirectOutput.jogForward := FALSE;
	  #statAxisIndexOld := #statActualAxisIndex;
	END_IF;
	
	#instLSimaHydTO_MC_RequestDirection(RequestForward := #hmiConnection.BasicAxisControl.Command.jogForward,
	                                    RequestBackward := #hmiConnection.BasicAxisControl.Command.jogBackward,
	                                    Axis := #axisData);
	
	
	CASE #hmiConnection.AxisSelector.Status.selectedTypeOfAxis OF
	    
	  2: // positioning axis
	    #instAxisBasicsPosAxis(axis := #hmiConnection.AxisSelector.Status.selectedTO_Axis,
	                           powerEnable := #hmiConnection.BasicAxisControl.Command.powerEnable,
	                           powerStartMode := #hmiConnection.BasicAxisControl.Command.powerStartMode,
	                           powerStopMode := #hmiConnection.BasicAxisControl.Command.powerStopMode,
	                           resetExecute := #hmiConnection.BasicAxisControl.Command.resetExecute,
	                           resetRestart := #hmiConnection.BasicAxisControl.Command.resetRestart,
	                           homeExecute := #hmiConnection.BasicAxisControl.Command.homeExecute,
	                           homePosition := #hmiConnection.BasicAxisControl.Command.homePosition,
	                           homeMode := #hmiConnection.BasicAxisControl.Command.homeMode,
	                           jogForward := #hmiConnection.BasicAxisControl.Command.jogForward AND #instLSimaHydTO_MC_RequestDirection.RampingForward,
	                           jogBackward := #hmiConnection.BasicAxisControl.Command.jogBackward AND #instLSimaHydTO_MC_RequestDirection.RampingBackward,
	                           jogVelocity := #hmiConnection.BasicAxisControl.Command.jogVelocity,
	                           jogAcceleration := #hmiConnection.BasicAxisControl.Command.jogAcceleration,
	                           jogDeceleration := #hmiConnection.BasicAxisControl.Command.jogDeceleration,
	                           jogJerk := #hmiConnection.BasicAxisControl.Command.jogJerk,
	                           jogPositionControlled := #hmiConnection.BasicAxisControl.Command.jogPositionControlled,
	                           powerStatus => #hmiConnection.BasicAxisControl.Status.powerStatus,
	                           powerBusy => #hmiConnection.BasicAxisControl.Status.powerBusy,
	                           resetDone => #hmiConnection.BasicAxisControl.Status.resetDone,
	                           resetBusy => #hmiConnection.BasicAxisControl.Status.resetBusy,
	                           homeDone => #hmiConnection.BasicAxisControl.Status.homeDone,
	                           homeBusy => #hmiConnection.BasicAxisControl.Status.homeBusy,
	                           jogInVelocity => #hmiConnection.BasicAxisControl.Status.jogInVelocity,
	                           jogBusy => #hmiConnection.BasicAxisControl.Status.jogBusy,
	                           commandAborted => #hmiConnection.BasicAxisControl.Status.commandAborted,
	                           error => #hmiConnection.BasicAxisControl.Status.error,
	                           errorID => #hmiConnection.BasicAxisControl.Status.errorID,
	                           statusID => #hmiConnection.BasicAxisControl.Status.statusID);
	    
	    #hmiConnection.AxisToData := "SimaHydTO_GetAxisToData_PosAxis"(#hmiConnection.AxisSelector.Status.selectedTO_Axis);
	    
	  3: // sync axis
	    #instAxisBasicsSyncAxis(axis := #hmiConnection.AxisSelector.Status.selectedTO_Axis,
	                            powerEnable := #hmiConnection.BasicAxisControl.Command.powerEnable,
	                            powerStartMode := #hmiConnection.BasicAxisControl.Command.powerStartMode,
	                            powerStopMode := #hmiConnection.BasicAxisControl.Command.powerStopMode,
	                            resetExecute := #hmiConnection.BasicAxisControl.Command.resetExecute,
	                            resetRestart := #hmiConnection.BasicAxisControl.Command.resetRestart,
	                            homeExecute := #hmiConnection.BasicAxisControl.Command.homeExecute,
	                            homePosition := #hmiConnection.BasicAxisControl.Command.homePosition,
	                            homeMode := #hmiConnection.BasicAxisControl.Command.homeMode,
	                            jogForward := #hmiConnection.BasicAxisControl.Command.jogForward,
	                            jogBackward := #hmiConnection.BasicAxisControl.Command.jogBackward,
	                            jogVelocity := #hmiConnection.BasicAxisControl.Command.jogVelocity,
	                            jogAcceleration := #hmiConnection.BasicAxisControl.Command.jogAcceleration,
	                            jogDeceleration := #hmiConnection.BasicAxisControl.Command.jogDeceleration,
	                            jogJerk := #hmiConnection.BasicAxisControl.Command.jogJerk,
	                            jogPositionControlled := #hmiConnection.BasicAxisControl.Command.jogPositionControlled,
	                            powerStatus => #hmiConnection.BasicAxisControl.Status.powerStatus,
	                            powerBusy => #hmiConnection.BasicAxisControl.Status.powerBusy,
	                            resetDone => #hmiConnection.BasicAxisControl.Status.resetDone,
	                            resetBusy => #hmiConnection.BasicAxisControl.Status.resetBusy,
	                            homeDone => #hmiConnection.BasicAxisControl.Status.homeDone,
	                            homeBusy => #hmiConnection.BasicAxisControl.Status.homeBusy,
	                            jogInVelocity => #hmiConnection.BasicAxisControl.Status.jogInVelocity,
	                            jogBusy => #hmiConnection.BasicAxisControl.Status.jogBusy,
	                            commandAborted => #hmiConnection.BasicAxisControl.Status.commandAborted,
	                            error => #hmiConnection.BasicAxisControl.Status.error,
	                            errorID => #hmiConnection.BasicAxisControl.Status.errorID,
	                            statusID => #hmiConnection.BasicAxisControl.Status.statusID);
	    
	    
	    #hmiConnection.AxisToData := "SimaHydTO_GetAxisToData_SyncAxis"(#hmiConnection.AxisSelector.Status.selectedTO_Axis);
	    
	  ELSE
	    ; // not suported
	    
	END_CASE;
	#hmiConnection.BasicAxisControl.ControlDirectOutput.safetyDistance := MAX(IN1 := 0.0, IN2 := #hmiConnection.BasicAxisControl.ControlDirectOutput.safetyDistance);
	#instDirectOutputControl(JogForward := #hmiConnection.BasicAxisControl.ControlDirectOutput.jogForward,
	                         JogBackward := #hmiConnection.BasicAxisControl.ControlDirectOutput.jogBackward,
	                         CommandValueForward := #hmiConnection.BasicAxisControl.ControlDirectOutput.commandValueForward,
	                         CommandValueBackward := #hmiConnection.BasicAxisControl.ControlDirectOutput.commandValueBackward,
	                         CommandValueRamp := #hmiConnection.BasicAxisControl.ControlDirectOutput.commandValueRamp,
	                         SafetyDistance := #hmiConnection.BasicAxisControl.ControlDirectOutput.safetyDistance,
	                         Busy => #hmiConnection.BasicAxisControl.StatusDirectOutput.active,
	                         MinSafetyPositionOverrun => #hmiConnection.BasicAxisControl.StatusDirectOutput.minSafetyPositionOverrun,
	                         MaxSafetyPositionOverrun => #hmiConnection.BasicAxisControl.StatusDirectOutput.maxSafetyPositionOverrun,
	                         Axis := #axisData);
	
	#instLSimaHydTO_MC_Reset(Execute:=#hmiConnection.BasicAxisControl.Command.resetFBExecute,
	                         Done=>#hmiConnection.BasicAxisControl.Status.resetFBDone,
	                         Busy=>#hmiConnection.BasicAxisControl.Status.resetFBBusy,
	                         Axis:=#axisData);
	
	
END_FUNCTION_BLOCK

FUNCTION_BLOCK "SimaHydTO_AxisBasics_SyncAxis"   // FB33193, FBD
TITLE = SimaHydTO_AxisBasics_SyncAxis
{ S7_Optimized_Access := 'TRUE' }
FAMILY : SimaHydTO/LAxisBasics
VERSION : 1.0
// Function block information: See Function block network 1
// stored: AutoNumber true, IsIECCheckEnabled false, IsRetainMemResEnabled false, MemoryReserve 100, SetENOAutomatically false, UDAEnableTagReadback false
   VAR_INPUT
      axis : TO_SynchronousAxis;   // Technology object (axis)
      powerEnable : Bool;   // MC_Power: 0: The technology object is disabled / 1: The technology object is enabled
      powerStartMode : DInt := 1;   // 0: Enable axis not position-controlled / 1: Enable axis position-controlled
      powerStopMode : Int := 0;   // 0: Emergency stop / 1: Immediate stop / 2: Stop with maximum dynamic values
      resetExecute : Bool;   // MC_Reset: Start job with a positive edge
      resetRestart : Bool := false;   // 0: Acknowledgment of queued technology alarms / 1: Reinitialization of the technology object and acknowledgment of pending technology alarms
      homeExecute : Bool;   // MC_Home: Start job with a positive edge
      homePosition : LReal;   // The specified value is used according to the selected "Mode".
      homeMode : Int;   // 0: Direct homing (absolute) / 1: Direct homing (relative) / 2: Passive homing / 3: Active homing / 4: Reserved / 5: Active homing (<TO>.Homing.HomePosition) / 6: Absolute encoder adjustment (relative) / 7: Absolute encoder adjustment (absolute) / 8: Passive homing / 9: Abort passive homing / 10: Passive homing (<TO>.Homing.HomePosition)
      jogForward : Bool;   // MC_MoveJog: As long as the parameter is TRUE, the axis moves in the positive direction
      jogBackward : Bool;   // MC_MoveJog: As long as the parameter is TRUE, the axis moves in the negative direction
      jogVelocity : LReal := 100.0;   // Velocity setpoint / speed setpoint for the motion
      jogAcceleration : LReal := -1.0;   // Acceleration of jog movement
      jogDeceleration : LReal := -1.0;   // Deceleration of jog movement
      jogJerk : LReal := -1.0;   // Jerk of jog movement
      jogPositionControlled : Bool := true;   // 0: Non position-controlled operation / 1: Position-controlled mode - The parameter applies as long as the MC_MoveJog command is executed. After this, the setting of MC_Power applies again.
   END_VAR
   VAR_OUTPUT
      powerStatus { ExternalWritable := 'False'} : Bool;   // MC_Power: 0: Technology object disabled / 1: Technology object enabled
      powerBusy { ExternalWritable := 'False'} : Bool;   // MC_Power: Job is running
      resetDone { ExternalWritable := 'False'} : Bool;   // MC_Reset: Error has been acknowledged or Restart has been executed.
      resetBusy { ExternalWritable := 'False'} : Bool;   // MC_Reset: Job is running
      homeDone { ExternalWritable := 'False'} : Bool;   // MC_Home: Job is completed
      homeBusy { ExternalWritable := 'False'} : Bool;   // MC_Home: Job is running
      jogInVelocity { ExternalWritable := 'False'} : Bool;   // MC_MoveJog: The velocity setpoint / speed setpoint was reached and will be maintained
      jogBusy { ExternalWritable := 'False'} : Bool;   // MC_MoveJog: Job is running
      commandAborted { ExternalWritable := 'False'} : Bool;   // The job was aborted by another job during execution (see also StatusID)
      error { ExternalWritable := 'False'} : Bool;   // An error occurred during execution of the job. The job is rejected. The cause of the error can be found in the "ErrorID" parameter.
      errorID { ExternalWritable := 'False'} : Word;   // ErrorID of motion control instruction (see also StatusID)
      statusID { ExternalWritable := 'False'} : Int;   // Additional specification of affected Motion control instruction of CommandAborted or Error: 0: No instruction / 1: MC_Power / 2: MC_Reset / 3: MC_Home / 4: MC_MoveJog
   END_VAR
   VAR
      instMcPower { ExternalAccessible := 'False'; ExternalVisible := 'False'; ExternalWritable := 'False'; S7_SetPoint := 'True'} : MC_POWER;   // PLCopen functions of basic motion control
      instMcReset { ExternalAccessible := 'False'; ExternalVisible := 'False'; ExternalWritable := 'False'; S7_SetPoint := 'True'} : MC_RESET;
      instMcHome { ExternalAccessible := 'False'; ExternalVisible := 'False'; ExternalWritable := 'False'; S7_SetPoint := 'True'} : MC_HOME;
      instMcMoveJog { ExternalAccessible := 'False'; ExternalVisible := 'False'; ExternalWritable := 'False'; S7_SetPoint := 'True'} : MC_MOVEJOG;
      statCommandAborted { ExternalAccessible := 'False'; ExternalVisible := 'False'; ExternalWritable := 'False'} : Array[#ARRAY_BEGIN..#ARRAY_END] of Bool;   // Arrays to save error information of PLCopen functions
      statError { ExternalAccessible := 'False'; ExternalVisible := 'False'; ExternalWritable := 'False'} : Array[#ARRAY_BEGIN..#ARRAY_END] of Bool;
      statErrorID { ExternalAccessible := 'False'; ExternalVisible := 'False'; ExternalWritable := 'False'} : Array[#ARRAY_BEGIN..#ARRAY_END] of Word;
   END_VAR
   VAR_TEMP
      tempDwordCommandAborted : DWord;   // Variables to check error informations of PLCopen functions
      tempDwordError : DWord;
      tempCount : Int;   // Counter of FOR counting loop
   END_VAR
   VAR CONSTANT
      ARRAY_BEGIN : Int := 1;   // Start-Index of array (Maximum 32 Array elements!)
      ARRAY_END : Int := 32;   // End-Index of array (Maximum 32 Array elements!)
      ERROR_DEFAULT : Bool := false;   // Default values of output signals
      ERRORID_DEFAULT : Word := 16#0;
      STATUSID_DEFAULT : Int := 0;
   END_VAR
BEGIN

REGION Network 1 (SCL): Axis Basics - Header
   //=============================================================================
   //SIEMENS AG
   //(c)Copyright 2016 All Rights Reserved
   //-----------------------------------------------------------------------------
   //Library:       AxisBasics
   //Tested with:   S7-1500 V2.5
   //Engineering:   TIA Portal V15
   //Restrictions:  Motion Control Library V4.0
   //Requirements:  S7-1500(T)
   //Functionality: Basic axis control of TO_SynchronousAxis
   //-----------------------------------------------------------------------------
   //Change log table:
   //Version  Date       Expert in charge Changes applied
   //01.00.00 04.10.2018 ArSc             First released version
   //=============================================================================
END_REGION

REGION Network 2: Axis Basics - MC_Power
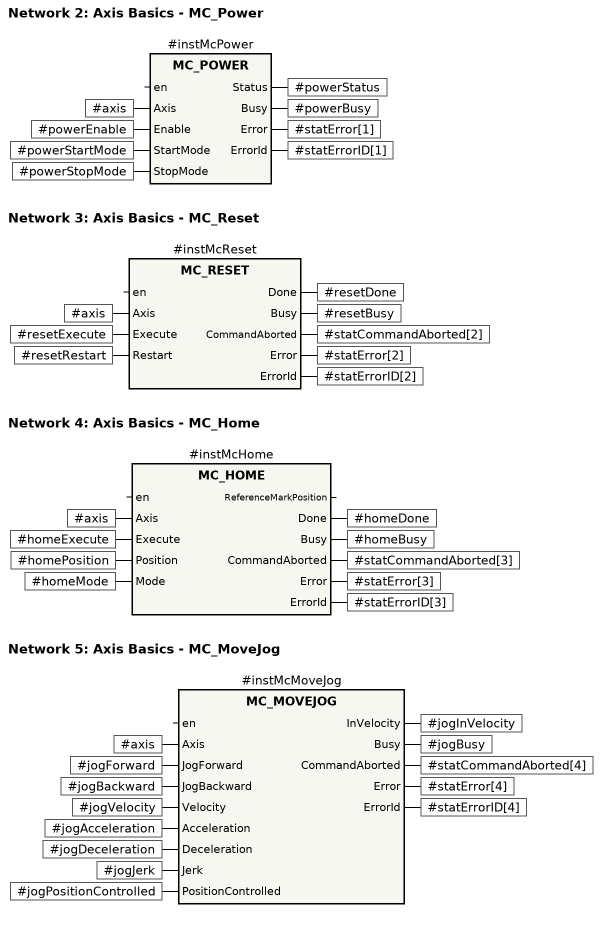
   #instMcPower(Axis := #axis,   // MC_POWER
                Enable := #powerEnable,
                StartMode := #powerStartMode,
                StopMode := #powerStopMode,
                Status => #powerStatus,
                Busy => #powerBusy,
                Error => #statError[1],
                ErrorId => #statErrorID[1]);
END_REGION

REGION Network 3: Axis Basics - MC_Reset
   #instMcReset(Axis := #axis,   // MC_RESET
                Execute := #resetExecute,
                Restart := #resetRestart,
                Done => #resetDone,
                Busy => #resetBusy,
                CommandAborted => #statCommandAborted[2],
                Error => #statError[2],
                ErrorId => #statErrorID[2]);
END_REGION

REGION Network 4: Axis Basics - MC_Home
   #instMcHome(Axis := #axis,   // MC_HOME
               Execute := #homeExecute,
               Position := #homePosition,
               Mode := #homeMode,
               Done => #homeDone,
               Busy => #homeBusy,
               CommandAborted => #statCommandAborted[3],
               Error => #statError[3],
               ErrorId => #statErrorID[3]);
END_REGION

REGION Network 5: Axis Basics - MC_MoveJog
   #instMcMoveJog(Axis := #axis,   // MC_MOVEJOG
                  JogForward := #jogForward,
                  JogBackward := #jogBackward,
                  Velocity := #jogVelocity,
                  Acceleration := #jogAcceleration,
                  Deceleration := #jogDeceleration,
                  Jerk := #jogJerk,
                  PositionControlled := #jogPositionControlled,
                  InVelocity => #jogInVelocity,
                  Busy => #jogBusy,
                  CommandAborted => #statCommandAborted[4],
                  Error => #statError[4],
                  ErrorId => #statErrorID[4]);
END_REGION

REGION Network 6 (SCL): Axis Basics - Generate output signals and error detection
   //General output signals

   //Reset output signals
   #commandAborted := False;
   #error := False;
   #errorID := #ERRORID_DEFAULT;
   #statusID := #STATUSID_DEFAULT;

   //Transfer ARRAY to DWORD
   GATHER(IN:=#statCommandAborted,
          OUT=>#tempDwordCommandAborted);
   GATHER(IN:=#statError,
          OUT=>#tempDwordError);

   //Check for errors or command aborts
   IF (#tempDwordError > DWORD#0)
   THEN
     //Select error information
     FOR #tempCount := #ARRAY_BEGIN TO #ARRAY_END
     DO
       IF (#statError[#tempCount] = True)
       THEN
         #error := True;
         #errorID := #statErrorID[#tempCount];
         #statusID := #tempCount;
         EXIT;
       END_IF;
     END_FOR;
   ELSIF (#tempDwordCommandAborted > DWORD#0)
   THEN
     //Select command aborted information
     FOR #tempCount := #ARRAY_BEGIN TO #ARRAY_END
     DO
       IF (#statCommandAborted[#tempCount] = True)
       THEN
         #commandAborted := True;
         #errorID := #statErrorID[#tempCount];
         #statusID := #tempCount;
         EXIT;
       END_IF;
     END_FOR;
   END_IF;
END_REGION
END_FUNCTION_BLOCK

FUNCTION_BLOCK "LSimaHydTO_MC_DirectOutputControl"
{ S7_Optimized_Access := 'TRUE' }
AUTHOR : APC_ERLF
FAMILY : LSimaHydTO
VERSION : 1.0
   VAR_INPUT 
      JogForward : Bool;
      JogBackward : Bool;
      CommandValueForward : LReal := 5.0;
      CommandValueBackward : LReal := 5.0;
      CommandValueRamp : LReal := 100.0;
      SafetyDistance : LReal := 50.0;
   END_VAR

   VAR_OUTPUT 
      CommandAborted { ExternalWritable := 'False'} : Bool;
      Busy { ExternalWritable := 'False'} : Bool;
      Error { ExternalWritable := 'False'} : Bool;
      ErrorID { ExternalWritable := 'False'} : Word;
      RampingDown { ExternalWritable := 'False'} : Bool;
      MinSafetyPositionOverrun { ExternalWritable := 'False'} : Bool;
      MaxSafetyPositionOverrun { ExternalWritable := 'False'} : Bool;
   END_VAR

   VAR_IN_OUT 
      Axis : "LSimaHydTO_typeAxisData";
   END_VAR

   VAR 
      statFBState { ExternalAccessible := 'False'; ExternalVisible := 'False'; ExternalWritable := 'False'} : DInt;
      statBusy { ExternalAccessible := 'False'; ExternalVisible := 'False'; ExternalWritable := 'False'} : Bool;
      statJigFwdOld { ExternalAccessible := 'False'; ExternalVisible := 'False'; ExternalWritable := 'False'} : Bool;
      statJogBkwdOld { ExternalAccessible := 'False'; ExternalVisible := 'False'; ExternalWritable := 'False'} : Bool;
   END_VAR

   VAR CONSTANT 
      FB_STATE_IDLE : DInt;
      FB_STATE_JOG : DInt := 10;
      FB_STATE_STOPPING : DInt := 20;
      FB_STATE_COMMAND_ABORTED : DInt := 30;
      FB_STATE_ERROR : DInt := -100;
      NO_ERROR_REACTION : DInt := 0;
      NO_ALARM : Word := 0;
      ALARM_AXIS_ERROR_OCCURED : Word := 16#8001;
      ALARM_WRONG_VALUE_VELOCITY : Word := 16#8003;
      ALARM_WRONG_VALUE_ACCEL : Word := 16#8004;
      ALARM_WRONG_DIRECTION : Word := 16#8007;
      ALARM_AXIS_DISABLED : Word := 16#800F;
   END_VAR


BEGIN
	//================================================================================
	//SIEMENS AG // (c)Copyright 2019 All Rights Reserved
	//--------------------------------------------------------------------------------
	//Library: LSimaHydTO
	//Tested with: S7-15xx
	//Engineering: TIA Portal  V15 (SW 2.5)
	//Restrictions: -
	//Requirements: S7-1500
	//Functionality:    controls the output of an axis directly according configuration
	//
	//--------------------------------------------------------------------------------
	//Change log table:
	//
	//Version     Date          Expert in charge    Changes applied
	//01.00.10    17.03.2018    APC_ERLF            First released version
	//================================================================================
	//
	REGION TRIGGERING
	  IF (#JogForward AND NOT #statJigFwdOld)
	    OR (#JogBackward AND NOT #statJogBkwdOld)
	  THEN
	    #CommandAborted := FALSE;
	    #statBusy := FALSE;
	    IF (#JogForward AND #Axis.Internal.Control.DirectOutput.commandValueForward <= 0.0) OR
	      (#JogBackward AND #Axis.Internal.Control.DirectOutput.commandValueBackward <= 0.0)
	    THEN
	      #Error := TRUE;
	      #ErrorID := #ALARM_WRONG_VALUE_VELOCITY;
	      #statFBState := #FB_STATE_ERROR;
	    ELSIF #Axis.Internal.Control.DirectOutput.commandValueRamp <= 0.0 THEN
	      #Error := TRUE;
	      #ErrorID := #ALARM_WRONG_VALUE_ACCEL;
	      #statFBState := #FB_STATE_ERROR;
	    ELSIF #JogForward AND #JogBackward THEN
	      #Error := TRUE;
	      #ErrorID := #ALARM_WRONG_DIRECTION;
	      #statFBState := #FB_STATE_ERROR;
	    ELSIF NOT #Axis.StatusActor.Enabled THEN
	      #Error := TRUE;
	      #ErrorID := #ALARM_AXIS_DISABLED;
	      #statFBState := #FB_STATE_ERROR;
	    ELSIF #Axis.ErrorDetail.Reaction <> #NO_ERROR_REACTION THEN
	      #Error := TRUE;
	      #ErrorID := #ALARM_AXIS_ERROR_OCCURED;
	      #statFBState := #FB_STATE_ERROR;
	    ELSE
	      #Axis.Internal.Control.DirectOutput.activate := TRUE;
	      #Axis.Internal.Control.DirectOutput.commandValueForward := #CommandValueForward;
	      #Axis.Internal.Control.DirectOutput.commandValueBackward := #CommandValueBackward;
	      #Axis.Internal.Control.DirectOutput.commandValueRamp := #CommandValueRamp;
	      #Axis.Internal.Control.DirectOutput.safetyDistance := #SafetyDistance;
	      #Axis.Internal.Control.DirectOutput.jogForward := #JogForward;
	      #Axis.Internal.Control.DirectOutput.jogBackward := #JogBackward;
	      
	      #statBusy := TRUE;
	      #Error := FALSE;
	      #ErrorID := #NO_ALARM;
	      #statFBState := #FB_STATE_JOG;
	    END_IF;
	    
	    
	  END_IF;
	  // Edge detection
	  #statJigFwdOld := #JogForward;
	  #statJogBkwdOld := #JogBackward;
	END_REGION
	
	IF #statFBState = #FB_STATE_IDLE THEN
	  RETURN;
	END_IF;
	
	REGION PRCESSING
	  IF #statBusy THEN
	    CASE #statFBState OF
	      #FB_STATE_JOG:
	        
	        IF NOT #Axis.StatusActor.Enabled OR #Axis.ErrorDetail.Reaction <> #NO_ERROR_REACTION THEN
	          #statBusy := FALSE;
	          #Error := TRUE;
	          IF #Axis.ErrorDetail.Reaction <> #NO_ERROR_REACTION THEN
	            #ErrorID := #ALARM_AXIS_ERROR_OCCURED;
	          ELSE
	            #ErrorID := #ALARM_AXIS_DISABLED;
	          END_IF;
	          #statFBState := #FB_STATE_ERROR;
	        ELSIF #Axis.Internal.MotionData.DirectOutput.rampingDown THEN
	          #Axis.Internal.Control.DirectOutput.jogForward := FALSE;
	          #Axis.Internal.Control.DirectOutput.jogBackward := FALSE;
	          
	          #statBusy := FALSE;
	          #CommandAborted := TRUE;
	          #statFBState := #FB_STATE_STOPPING;
	        ELSE
	          #Axis.Internal.Control.DirectOutput.jogForward := #JogForward;
	          #Axis.Internal.Control.DirectOutput.jogBackward := #JogBackward;
	          
	          IF NOT (#JogForward OR #JogBackward) THEN
	            
	            #statFBState := #FB_STATE_STOPPING;
	          END_IF;
	        END_IF;
	      #FB_STATE_STOPPING:
	        IF NOT #Axis.Internal.MotionData.DirectOutput.active THEN
	          #Axis.Internal.Control.DirectOutput.activate := FALSE;
	          #statBusy := FALSE;
	          #statFBState := #FB_STATE_IDLE;
	        END_IF;
	    END_CASE;
	  END_IF;
	END_REGION
	REGION OUTPUTS
	  
	  CASE #statFBState OF
	      
	    #FB_STATE_COMMAND_ABORTED:
	      IF NOT (#JogForward OR #JogBackward) THEN
	        #statBusy := FALSE;
	        #CommandAborted := FALSE;
	        
	        #statFBState := #FB_STATE_IDLE;
	      END_IF;
	      
	      
	    #FB_STATE_ERROR:
	      IF NOT (#JogForward OR #JogBackward) THEN
	        #statFBState := #FB_STATE_IDLE;
	        #Error := FALSE;
	        #ErrorID := #NO_ALARM;
	      END_IF;
	  END_CASE;
	  #RampingDown := #Axis.Internal.MotionData.DirectOutput.rampingDown;
	  #MinSafetyPositionOverrun := #Axis.Internal.MotionData.DirectOutput.minSafetyPositionOverrun;
	  #MaxSafetyPositionOverrun := #Axis.Internal.MotionData.DirectOutput.maxSafetyPositionOverrun;
	  #Busy := #statBusy;
	  IF #statFBState = #FB_STATE_IDLE THEN
	    #Axis.Internal.Control.DirectOutput.jogForward := FALSE;
	    #Axis.Internal.Control.DirectOutput.jogBackward := FALSE;
	    #Axis.Internal.Control.DirectOutput.activate := FALSE;
	    #statBusy := #Busy := #CommandAborted := #Error := #RampingDown := #MinSafetyPositionOverrun := #MaxSafetyPositionOverrun := FALSE;
	    #ErrorID := #NO_ALARM;
	  END_IF;
	END_REGION
END_FUNCTION_BLOCK

FUNCTION_BLOCK "LSimaHydTO_MC_RequestDirection"
{ S7_Optimized_Access := 'TRUE' }
AUTHOR : APC_ERLF
FAMILY : LSimaHydTO
VERSION : 1.0
   VAR_INPUT 
      RequestForward : Bool;
      RequestBackward : Bool;
   END_VAR

   VAR_OUTPUT 
      ValveForward { ExternalWritable := 'False'} : Bool := FALSE;
      ValveBackward { ExternalWritable := 'False'} : Bool := FALSE;
      RampingForward { ExternalWritable := 'False'} : Bool;
      RampingBackward { ExternalWritable := 'False'} : Bool;
      Busy { ExternalWritable := 'False'} : Bool;
      CommandAborted { ExternalWritable := 'False'} : Bool;
      Error { ExternalWritable := 'False'} : Bool;
      ErrorID { ExternalWritable := 'False'} : Word;
   END_VAR

   VAR_IN_OUT 
      Axis : "LSimaHydTO_typeAxisData";
   END_VAR

   VAR 
      statFBState { ExternalAccessible := 'False'; ExternalVisible := 'False'; ExternalWritable := 'False'} : SInt;
      statReqFwdOld { ExternalAccessible := 'False'; ExternalVisible := 'False'; ExternalWritable := 'False'} : Bool;
      statReqBackOld { ExternalAccessible := 'False'; ExternalVisible := 'False'; ExternalWritable := 'False'} : Bool;
      statExecuteOld { ExternalAccessible := 'False'; ExternalVisible := 'False'; ExternalWritable := 'False'} : Bool;
   END_VAR

   VAR_TEMP 
      tempExecute : Bool;
   END_VAR

   VAR CONSTANT 
      STATE_IDLE : SInt;
      STATE_MOVEMENT : SInt := 10;
      STATE_STOPPING : SInt := 20;
      STATE_COMMAND_ABORTED : SInt := 30;
      STATE_ERROR : SInt := -100;
      NO_ERROR_REACTION : DInt := 0;
      NO_ALARM : Word := 0;
      ALARM_AXIS_ERROR_OCCURED : Word := 16#8001;
      ALARM_WRONG_DIRECTION : Word := 16#8007;
      ALARM_AXIS_DISABLED : Word := 16#800F;
   END_VAR


BEGIN
	//================================================================================
	//SIEMENS AG // (c)Copyright 2019 All Rights Reserved
	//--------------------------------------------------------------------------------
	//Library: LSimaHydTO
	//Tested with: S7-15xx
	//Engineering: TIA Portal  V15 (SW 2.5)
	//Restrictions: -
	//Requirements: S7-1500
	//Functionality:    request switching direction valves and recognize the enabling of motion control
	//
	//--------------------------------------------------------------------------------
	//Change log table:
	//
	//Version     Date          Expert in charge    Changes applied
	//01.00.00    11.09.2019    APC_ERLF            First released version
	//================================================================================
	
	#tempExecute := (#RequestForward AND NOT #statReqFwdOld)
	             OR (#RequestBackward AND NOT #statReqBackOld);
	             
	//
	IF #tempExecute AND NOT #statExecuteOld THEN
	  #CommandAborted := FALSE;
	  #Busy := FALSE;
	  IF #RequestForward AND #RequestBackward THEN
	    #Error := TRUE;
	    #ErrorID := #ALARM_WRONG_DIRECTION;
	    #statFBState := #STATE_ERROR;
	  ELSIF NOT #Axis.StatusActor.Enabled THEN
	    #Error := TRUE;
	    #ErrorID := #ALARM_AXIS_DISABLED;
	    #statFBState := #STATE_ERROR;
	  ELSIF #Axis.ErrorDetail.Reaction <> #NO_ERROR_REACTION THEN
	    #Error := TRUE;
	    #ErrorID := #ALARM_AXIS_ERROR_OCCURED;
	    #statFBState := #STATE_ERROR;
	  ELSE
	    #Axis.Internal.Control.RequestForward := #RequestForward;
	    #Axis.Internal.Control.RequestBackward := #RequestBackward;
	    
	    #Busy := TRUE;
	    #Error := FALSE;
	    #ErrorID := #NO_ALARM;
	    #statFBState := #STATE_MOVEMENT;
	  END_IF;
	END_IF;
	 
	
	#statReqFwdOld := #RequestForward;
	#statReqBackOld := #RequestBackward;
	#statExecuteOld := #tempExecute;
	             
	             
	
	  CASE #statFBState OF
	    #STATE_IDLE:  // Idle
	      ;
	      
	    #STATE_MOVEMENT:
	      
	      IF NOT #Axis.StatusActor.Enabled OR #Axis.ErrorDetail.Reaction <> #NO_ERROR_REACTION THEN
	        #Busy := FALSE;
	        #Error := TRUE;
	        IF #Axis.ErrorDetail.Reaction <> #NO_ERROR_REACTION THEN
	          #ErrorID := #ALARM_AXIS_ERROR_OCCURED;
	        ELSE
	          #ErrorID := #ALARM_AXIS_DISABLED;
	        END_IF;
	        #statFBState := #STATE_ERROR;
	      ELSIF NOT (#RequestForward OR #RequestBackward) THEN
	          #Axis.Internal.Control.RequestForward := FALSE;
	          #Axis.Internal.Control.RequestBackward := FALSE;
	          
	          #statFBState := #STATE_IDLE;
	          
	        
	      ELSIF     #Axis.Internal.Control.RequestForward <> #RequestForward
	        OR  #Axis.Internal.Control.RequestBackward <> #RequestBackward
	      THEN
	        
	        #Busy := FALSE;
	        #CommandAborted := TRUE;
	        #statFBState := #STATE_COMMAND_ABORTED;
	      END_IF;
	  END_CASE;
	  
	  CASE #statFBState OF
	      
	    #STATE_COMMAND_ABORTED:
	      IF NOT (#RequestForward OR #RequestBackward) THEN
	        #CommandAborted := FALSE;
	        
	        #statFBState := #STATE_IDLE;
	      END_IF;
	      
	    #STATE_ERROR:
	      IF NOT (#RequestForward OR #RequestBackward) THEN
	        #statFBState := #STATE_IDLE;
	        #Error := FALSE;
	        #ErrorID := #NO_ALARM;
	      END_IF;
	  END_CASE;
	  
	  // write outputs
	  #ValveForward := #Axis.StatusActor.ValveForward;
	  #ValveBackward := #Axis.StatusActor.ValveBackward;
	  #RampingForward := #Axis.Internal.MotionData.RampingForward;
	  #RampingBackward := #Axis.Internal.MotionData.RampingBackward;
	  
END_FUNCTION_BLOCK

FUNCTION_BLOCK "LSimaHydTO_MC_Reset"
{ S7_Optimized_Access := 'TRUE' }
AUTHOR : APC_ERLF
FAMILY : LSimaHydTO
VERSION : 1.0
   VAR_INPUT 
      Execute : Bool;
   END_VAR

   VAR_OUTPUT 
      Done { ExternalWritable := 'False'} : Bool;
      Busy { ExternalWritable := 'False'} : Bool;
      CommandAborted { ExternalWritable := 'False'} : Bool;
      Error { ExternalWritable := 'False'} : Bool;
      ErrorID { ExternalWritable := 'False'} : Word;
   END_VAR

   VAR_IN_OUT 
      Axis : "LSimaHydTO_typeAxisData";
   END_VAR

   VAR 
      statFBState { ExternalAccessible := 'False'; ExternalVisible := 'False'; ExternalWritable := 'False'} : DInt;
      statExecuteOld { ExternalAccessible := 'False'; ExternalVisible := 'False'; ExternalWritable := 'False'} : Bool;
   END_VAR

   VAR CONSTANT 
      NO_ERROR : Word := 16#0000_0000;
      STATE_IDLE : DInt;
      STATE_FIRST_CYCLE : DInt := 10;
      STATE_BUSY : DInt := 20;
      STATE_DONE : DInt := 30;
      STATE_COMMAND_ABORTED : DInt := 40;
      STATE_ERROR : DInt := 100;
   END_VAR


BEGIN
	//================================================================================
	//SIEMENS AG // (c)Copyright 2016 All Rights Reserved
	//--------------------------------------------------------------------------------
	//Library: LSimaHydTO
	//Tested with: S7-15xx
	//Engineering: TIA Portal  V15 (SW 2.5)
	//Restrictions: -
	//Requirements: S7-1500
	//Functionality:    acknowledges all technology alarms that can be acknowledged 
	//                  in the user program
	//
	//-------------------------------------------------------------------------------9
	//Change log table:
	//
	//Version     Date          Expert in charge    Changes applied
	//01.00.00    15.03.2018    APC_ERLF            First released version
	//================================================================================
	
	
	// ----------------------------------------------------------------------
	// start
	// ----------------------------------------------------------------------
	// rising edge of execute starts functionality
	IF #Execute AND NOT #statExecuteOld  THEN
	    // initialization
	    #Done := FALSE;
	    #CommandAborted := FALSE;
	    #Busy := FALSE;
	    #Error := FALSE;
	    #ErrorID := #NO_ERROR;
	    #statFBState := #STATE_FIRST_CYCLE;
	END_IF;
	
	// ----------------------------------------------------------------------
	// busy
	// ----------------------------------------------------------------------
	  CASE #statFBState OF
	    #STATE_FIRST_CYCLE:
	      
	      #CommandAborted := FALSE;
	      #Axis.Internal.Control.AckError := TRUE;
	      
	      IF   #Axis.ErrorWord = 0  THEN
	        #Done := TRUE;
	          #statFBState := #STATE_DONE;
	          
	        ELSE
	            #Busy := TRUE;
	            #statFBState := #STATE_BUSY;
	        END_IF;
	        
	      
	      #STATE_BUSY:
	        
	        IF #Axis.ErrorWord = 0 THEN
	          #Axis.Internal.Control.AckError := FALSE;
	          
	          #Done := TRUE;
	          #Busy := FALSE;
	          #statFBState := #STATE_DONE;
	          
	        END_IF;
	      
	// -------------------------------------------------------------------------
	// state analysis (no function)
	// -------------------------------------------------------------------------
	  #STATE_IDLE:
	    // ======================================================================
	    ;
	    
	  #STATE_DONE:
	    // ======================================================================
	    // output for one cycle minimum
	    // 
	    IF #Axis.ErrorWord = 0 THEN
	      #Axis.Internal.Control.AckError := FALSE;
	    END_IF;
	    IF NOT #Execute THEN
	      #Done := FALSE;
	      #Axis.Internal.Control.AckError := FALSE;
	      #statFBState := #STATE_IDLE;
	    END_IF;
	    
	  #STATE_COMMAND_ABORTED:
	    // ======================================================================
	    // reset commandAborted, output for one cycle minimum
	    IF NOT #Execute THEN
	      #CommandAborted := FALSE;
	      #statFBState := #STATE_IDLE;
	    END_IF;
	    
	  #STATE_ERROR:
	    // ======================================================================
	    // reset error, output for one cycle minimum
	    IF #Axis.ErrorWord = 0 THEN
	      #Axis.Internal.Control.AckError := FALSE;
	    END_IF;
	    IF NOT #Execute THEN
	      #Axis.Internal.Control.AckError := FALSE;
	      #Error := FALSE;
	      #ErrorID := #NO_ERROR;
	      #statFBState := #STATE_IDLE;
	    END_IF;
	    
	    
	  ELSE
	    // ======================================================================
	    // when FB is busy...
	    ;
	END_CASE;
	
	// -------------------------------------------------------------------------
	// always executed
	// -------------------------------------------------------------------------
	
	// edge detection
	#statExecuteOld := #Execute;
	
	
END_FUNCTION_BLOCK

FUNCTION "SimaHydTO_GetAxisToData_PosAxis" : "SimaHydTO_typeHMIConnectionAxisToData"
{ S7_Optimized_Access := 'TRUE' }
FAMILY : SimaHydTO
VERSION : 1.0
   VAR_INPUT 
      axisTO {InstructionName := 'TO_PositioningAxis'; LibVersion := '4.0'} : TO_PositioningAxis;
   END_VAR


BEGIN
	//=============================================================================
	//SIEMENS AG
	//(c)Copyright 2016 All Rights Reserved
	//-----------------------------------------------------------------------------
	//Library:       SimaHyd_AxisBasics
	//Tested with:   S7-1500 V2.5
	//Engineering:   TIA Portal V15
	//Restrictions:  Motion Control Library V4.0
	//Requirements:  S7-1500(T)
	//Functionality: Get axis data of TO_PositioningAxis
	//-----------------------------------------------------------------------------
	//Change log table:
	//Version  Date       Expert in charge Changes applied
	//01.00.00 20.05.2019 ArSc             First released version
	//=============================================================================
	
	
	//-----------------------------------------------------------------------------
	//Write axis data
	//-----------------------------------------------------------------------------
	#SimaHydTO_GetAxisToData_PosAxis.statusWord := #axisTO.StatusWord;
	#SimaHydTO_GetAxisToData_PosAxis.warningWord := #axisTO.WarningWord;
	#SimaHydTO_GetAxisToData_PosAxis.errorWord := #axisTO.ErrorWord;
	#SimaHydTO_GetAxisToData_PosAxis.errorDetail.number := #axisTO.ErrorDetail.Number;
	#SimaHydTO_GetAxisToData_PosAxis.errorDetail.reaction := #axisTO.ErrorDetail.Reaction;
	
	
END_FUNCTION

FUNCTION "SimaHydTO_GetAxisToData_SyncAxis" : "SimaHydTO_typeHMIConnectionAxisToData"
{ S7_Optimized_Access := 'TRUE' }
FAMILY : SimaHydTO
VERSION : 1.0
   VAR_INPUT 
      axisTO {InstructionName := 'TO_SynchronousAxis'; LibVersion := '4.0'} : TO_SynchronousAxis;
   END_VAR


BEGIN
	//=============================================================================
	//SIEMENS AG
	//(c)Copyright 2016 All Rights Reserved
	//-----------------------------------------------------------------------------
	//Library:       SimaHyd_AxisBasics
	//Tested with:   S7-1500 V2.5
	//Engineering:   TIA Portal V15
	//Restrictions:  Motion Control Library V4.0
	//Requirements:  S7-1500(T)
	//Functionality: Get axis data of TO_SynchronousAxis
	//-----------------------------------------------------------------------------
	//Change log table:
	//Version  Date       Expert in charge Changes applied
	//01.00.00 20.05.2019 ArSc             First released version
	//=============================================================================
	
	
	//-----------------------------------------------------------------------------
	//Write axis data
	//-----------------------------------------------------------------------------
	#SimaHydTO_GetAxisToData_SyncAxis := "SimaHydTO_GetAxisToData_PosAxis"(#axisTO);
END_FUNCTION

FUNCTION_BLOCK "SimaHydTO_VCharMeasurement"
{ S7_Optimized_Access := 'TRUE' }
FAMILY : SimaHydTO
VERSION : 1.0
   VAR_IN_OUT 
      hmiConnection : "SimaHydTO_typeHMIConnection";
      axisData : "LSimaHydTO_typeAxisData";
      axesArray : Array[*] of "SimaHydTO_typeAxesArray";
      vCharArray : Array[*] of "SimaHydTO_typeVCharArray";
   END_VAR

   VAR 
      statFirstRunDone { ExternalAccessible := 'False'; ExternalVisible := 'False'; ExternalWritable := 'False'} : Bool;
      statActualAxisDB { ExternalAccessible := 'False'; ExternalVisible := 'False'; ExternalWritable := 'False'} : DB_ANY;
      statActualVCharIndex { ExternalAccessible := 'False'; ExternalVisible := 'False'; ExternalWritable := 'False'} : Int;
      statVCharIndexOld { ExternalAccessible := 'False'; ExternalVisible := 'False'; ExternalWritable := 'False'} : Int := -1;
      statExecute { ExternalAccessible := 'False'; ExternalVisible := 'False'; ExternalWritable := 'False'} : Bool;
      statContinue { ExternalAccessible := 'False'; ExternalVisible := 'False'; ExternalWritable := 'False'} : Bool;
      statExecuteOld { ExternalAccessible := 'False'; ExternalVisible := 'False'; ExternalWritable := 'False'} : Bool;
      instGetCharacteristics { ExternalAccessible := 'False'; ExternalVisible := 'False'; ExternalWritable := 'False'} : "LSimaHydTO_GetCharacteristic";
      instHmiVCharSelector { ExternalAccessible := 'False'; ExternalVisible := 'False'; ExternalWritable := 'False'} : "SimaHydTO_HmiVCharSelector";
      statLoadOld { ExternalAccessible := 'False'; ExternalVisible := 'False'; ExternalWritable := 'False'} : Bool;
      statSaveOld { ExternalAccessible := 'False'; ExternalVisible := 'False'; ExternalWritable := 'False'} : Bool;
      statSaveToDBL { ExternalAccessible := 'False'; ExternalVisible := 'False'; ExternalWritable := 'False'} : Bool;
      statBusyWrite { ExternalAccessible := 'False'; ExternalVisible := 'False'; ExternalWritable := 'False'} : Bool;
      statRampigForward { ExternalAccessible := 'False'; ExternalVisible := 'False'; ExternalWritable := 'False'} : Bool;
      statRampingBackward { ExternalAccessible := 'False'; ExternalVisible := 'False'; ExternalWritable := 'False'} : Bool;
      statActualAxisIndex { ExternalAccessible := 'False'; ExternalVisible := 'False'; ExternalWritable := 'False'} : Int;
      statVCharArrMinIndex { ExternalAccessible := 'False'; ExternalVisible := 'False'; ExternalWritable := 'False'} : Int;
      statVCharArrMaxIndex { ExternalAccessible := 'False'; ExternalVisible := 'False'; ExternalWritable := 'False'} : Int;
      statDefaultConfig { ExternalAccessible := 'False'; ExternalVisible := 'False'; ExternalWritable := 'False'} : "LSimaHydTO_typeMeasurementConfig";
   END_VAR

   VAR_TEMP 
      tempVariant : Variant;
      tempHydAxis : REF_TO "LSimaHydTO_typeAxisData";
      tempErrorVariant : Int;
      tempRetVal : Int;
      tempInt : Int;
      tempSearchDone : Bool;
   END_VAR


BEGIN
	//=============================================================================
	//SIEMENS AG
	//(c)Copyright 2016 All Rights Reserved
	//-----------------------------------------------------------------------------
	//Library:       SimaHydTO_VCharMeasurement
	//Tested with:   S7-1500 V2.5
	//Engineering:   TIA Portal V15
	//Restrictions:  -
	//Requirements:  S7-1500(T)
	//Functionality: Automatic measurement of valve characteristics
	//-----------------------------------------------------------------------------
	//Change log table:
	//Version  Date       Expert in charge Changes applied
	//01.00.00 16.07.2019 ArSc             First released version
	//=============================================================================
	
	//Array detection and initialization
	IF (#statFirstRunDone = False)
	THEN
	  //Get MIN and MAX of array indices
	  #statVCharArrMinIndex := DINT_TO_INT(LOWER_BOUND(ARR := #vCharArray, DIM := 1));
	  #statVCharArrMaxIndex := DINT_TO_INT(UPPER_BOUND(ARR := #vCharArray, DIM := 1));
	  //Set default value of actual axis index
	  #statActualVCharIndex := #statVCharArrMinIndex - 1;
	  #statVCharIndexOld := #statActualVCharIndex;
	  
	  //Mark first run of function block
	  #statFirstRunDone := True;
	END_IF;
	
	(*
	  #instHmiVCharSelector(command := #hmiConnection.VCharEditor.Command.VCharLoad,
	                         status => #hmiConnection.VCharEditor.Status.VCharLoad,
	                         VCharArray := #VCharArray);
	                         *)
	
	//Check axis selection, if axis has changed
	IF #hmiConnection.AxisSelector.Status.selectionChanged
	  AND #hmiConnection.AxisSelector.Status.dataValid
	THEN
	  
	  #statActualAxisIndex := #hmiConnection.AxisSelector.Status.actualAxisIndex;
	  #tempSearchDone := FALSE;
	  FOR #tempInt := #statVCharArrMinIndex TO #statVCharArrMaxIndex DO
	    IF #vCharArray[#tempInt].VChar_DB = #hmiConnection.AxisSelector.Status.selectedVChar THEN
	      #statActualVCharIndex := #tempInt;
	      #tempSearchDone := TRUE;
	      EXIT;
	    END_IF;
	  END_FOR;
	  IF NOT #tempSearchDone THEN
	    #statActualVCharIndex := #statVCharArrMinIndex - 1;
	  END_IF;
	  
	END_IF;
	
	IF  #hmiConnection.GetCharacteristics.Command.loadConfig AND NOT #statLoadOld 
	  THEN
	    IF #statActualVCharIndex >= #statVCharArrMinIndex THEN
	      #hmiConnection.GetCharacteristics.ConfigData := #vCharArray[#statActualVCharIndex].measurementConfig;
	      #hmiConnection.BasicAxisControl.ControlDirectOutput.safetyDistance := #hmiConnection.GetCharacteristics.ConfigData.safetyDistance;
	      #hmiConnection.GetCharacteristics.Command.abort := FALSE;
	      #hmiConnection.GetCharacteristics.Command.execute := FALSE;
	      #hmiConnection.GetCharacteristics.Command.saveConfig := FALSE;
	      #hmiConnection.GetCharacteristics.Command.loadConfig := FALSE;
	    ELSE
	      #hmiConnection.GetCharacteristics.ConfigData := #statDefaultConfig;
	    END_IF;
	    #statVCharIndexOld := #statActualVCharIndex;
	    
	  END_IF;
	  
	//Check start of measurement
	IF (#hmiConnection.GetCharacteristics.Command.execute
	  AND NOT #statExecuteOld
	  AND NOT #hmiConnection.GetCharacteristics.Status.busy
	  AND #hmiConnection.AxisSelector.Status.dataValid)
	THEN
	  //Save axis selection
	  
	  #statActualAxisDB := #hmiConnection.AxisSelector.Status.selectedAxis;
	  #statActualAxisIndex := #hmiConnection.AxisSelector.Status.actualAxisIndex;
	  #hmiConnection.GetCharacteristics.ConfigData.safetyDistance := #hmiConnection.BasicAxisControl.ControlDirectOutput.safetyDistance;
	  IF #statActualVCharIndex >= #statVCharArrMinIndex THEN
	    #vCharArray[#statActualVCharIndex].measurementConfig := #hmiConnection.GetCharacteristics.ConfigData;
	  END_IF;
	  
	  #statExecute := TRUE;
	ELSIF(#hmiConnection.GetCharacteristics.Command.execute
	  AND NOT #statExecuteOld
	  AND #hmiConnection.GetCharacteristics.Status.busy)
	THEN
	  #statContinue := TRUE;
	END_IF;
	
	//Do measurement
	IF #hmiConnection.GetCharacteristics.Status.busy THEN
	  #statRampigForward := #axesArray[#statActualAxisIndex].VCharMeasurement.enableRampingForward;
	  #statRampingBackward := #axesArray[#statActualAxisIndex].VCharMeasurement.enableRampingBackward;
	  
	END_IF;
	#tempVariant := DB_ANY_TO_VARIANT(in := #statActualAxisDB, err => #tempErrorVariant);
	
	IF TypeOf(#tempVariant) = LSimaHydTO_typeAxisData THEN
	  //Get hydraulic axis data
	  #tempHydAxis ?= #tempVariant;
	  //Call measurement function block
	  #instGetCharacteristics(execute:=#statExecute,
	                          abort:=#hmiConnection.GetCharacteristics.Command.abort,
	                          continueMeasurement:=#statContinue,
	                          enableRampingForward:=#hmiConnection.GetCharacteristics.Command.enableRampingForward AND #statRampigForward,
	                          enableRampingBackward:=#hmiConnection.GetCharacteristics.Command.enableRampingBackward AND #statRampingBackward,
	                          qOutputValueStepForward=>#hmiConnection.GetCharacteristics.Status.qOutputValueStepForward,
	                          qOutputValueStepBackward=>#hmiConnection.GetCharacteristics.Status.qOutputValueStepBackward,
	                          velocityStepForward=>#hmiConnection.GetCharacteristics.Status.velocityStepForward,
	                          velocityStepBackward=>#hmiConnection.GetCharacteristics.Status.velocityStepBackward,
	                          requestForward=>#hmiConnection.GetCharacteristics.Status.requestForward,
	                          requestBackward=>#hmiConnection.GetCharacteristics.Status.requestBackward,
	                          statusMeasurement=>#hmiConnection.GetCharacteristics.Status.statusMeasurement,
	                         // done=>#hmiConnection.GetCharacteristics.Status.done,
	                          busy=>#hmiConnection.GetCharacteristics.Status.busy,
	                         // commandAborted=>#hmiConnection.GetCharacteristics.Status.commandAborted,
	                         // error=>#hmiConnection.GetCharacteristics.Status.error,
	                         // status=>#hmiConnection.GetCharacteristics.Status.status,
	                          measuredValues := #hmiConnection.GetCharacteristics.MeasuredValues,
	                          configData := #hmiConnection.GetCharacteristics.ConfigData,
	                          axis := #tempHydAxis^);
	  
	  #axesArray[#statActualAxisIndex].VCharMeasurement.requestForward := #hmiConnection.GetCharacteristics.Status.requestForward;
	  #axesArray[#statActualAxisIndex].VCharMeasurement.requestBackward := #hmiConnection.GetCharacteristics.Status.requestBackward;
	  
	  IF #instGetCharacteristics.error THEN
	    #hmiConnection.GetCharacteristics.Status.error := TRUE;
	    #hmiConnection.GetCharacteristics.Status.done := FALSE;
	    #hmiConnection.GetCharacteristics.Status.commandAborted := FALSE;
	  ELSIF #instGetCharacteristics.commandAborted THEN
	    #hmiConnection.GetCharacteristics.Status.commandAborted := TRUE;
	    #hmiConnection.GetCharacteristics.Status.done := FALSE;
	  ELSIF #instGetCharacteristics.done THEN
	    #hmiConnection.GetCharacteristics.Status.done := TRUE;
	  ELSIF #instGetCharacteristics.busy THEN
	    #hmiConnection.GetCharacteristics.Status.done := FALSE;
	    #hmiConnection.GetCharacteristics.Status.commandAborted := FALSE;
	    #hmiConnection.GetCharacteristics.Status.error := FALSE;
	  END_IF;
	    
	  IF #instGetCharacteristics.status <> 16#7000 OR NOT (#hmiConnection.GetCharacteristics.Status.error OR #hmiConnection.GetCharacteristics.Status.commandAborted)
	  THEN
	    #hmiConnection.GetCharacteristics.Status.status := #instGetCharacteristics.status;
	  END_IF;
	  
	END_IF;
	
	// save configuration
	IF #hmiConnection.GetCharacteristics.Command.saveConfig
	  AND NOT #statSaveOld
	  AND #statActualVCharIndex >= #statVCharArrMinIndex
	THEN
	  #vCharArray[#statActualVCharIndex].measurementConfig := #hmiConnection.GetCharacteristics.ConfigData;
	  #statSaveToDBL := TRUE;
	END_IF;
	
	IF #statSaveToDBL THEN
	  #tempRetVal := WRIT_DBL(REQ := TRUE,
	                          SRCBLK := #vCharArray[#statActualVCharIndex],
	                          BUSY => #statBusyWrite,
	                          DSTBLK => #vCharArray[#statActualVCharIndex]);
	  IF NOT #statBusyWrite THEN
	    #statSaveToDBL := FALSE;
	  END_IF;
	  
	END_IF;
	
	#statExecute := FALSE;
	#statContinue := FALSE;
	//Save data from last cycle
	#statExecuteOld := #hmiConnection.GetCharacteristics.Command.execute;
	#statSaveOld := #hmiConnection.GetCharacteristics.Command.saveConfig;
	#statLoadOld := #hmiConnection.GetCharacteristics.Command.loadConfig;
	
END_FUNCTION_BLOCK

FUNCTION_BLOCK "LSimaHydTO_GetCharacteristic"
{ S7_Optimized_Access := 'TRUE' }
AUTHOR : APC_ERLF
FAMILY : LSimaHydTO
VERSION : 1.22
   VAR_INPUT 
      execute : Bool;
      abort : Bool;
      continueMeasurement : Bool;
      enableRampingForward : Bool;
      enableRampingBackward : Bool;
   END_VAR

   VAR_OUTPUT 
      qOutputValueStepForward { ExternalWritable := 'False'} : LReal;
      qOutputValueStepBackward { ExternalWritable := 'False'} : LReal;
      velocityStepForward { ExternalWritable := 'False'} : LReal;
      velocityStepBackward { ExternalWritable := 'False'} : LReal;
      requestForward { ExternalWritable := 'False'} : Bool;
      requestBackward { ExternalWritable := 'False'} : Bool;
      statusMeasurement { ExternalWritable := 'False'} : Word;
      done { ExternalWritable := 'False'} : Bool;
      busy { ExternalWritable := 'False'} : Bool;
      commandAborted { ExternalWritable := 'False'} : Bool;
      error { ExternalWritable := 'False'} : Bool;
      status { ExternalWritable := 'False'} : Word;
   END_VAR

   VAR_IN_OUT 
      measuredValues : "LSimaHydTO_typeMeasuredValues";
      configData : "LSimaHydTO_typeMeasurementConfig";
      axis : "LSimaHydTO_typeAxisData";
   END_VAR

   VAR 
      statExecuteOld { ExternalAccessible := 'False'; ExternalVisible := 'False'; ExternalWritable := 'False'} : Bool;
      statDone { ExternalAccessible := 'False'; ExternalVisible := 'False'; ExternalWritable := 'False'} : Bool;
      statBusy { ExternalAccessible := 'False'; ExternalVisible := 'False'; ExternalWritable := 'False'} : Bool;
      statError { ExternalAccessible := 'False'; ExternalVisible := 'False'; ExternalWritable := 'False'} : Bool;
      statStatus { ExternalAccessible := 'False'; ExternalVisible := 'False'; ExternalWritable := 'False'} : Word := #STATUS_NO_CALL;
      statFBState { ExternalAccessible := 'False'; ExternalVisible := 'False'; ExternalWritable := 'False'} : DInt := #FB_STATE_NO_PROCESSING;
      statFBStateOld { ExternalAccessible := 'False'; ExternalVisible := 'False'; ExternalWritable := 'False'} : DInt := #FB_STATE_NO_PROCESSING;
      statNumOfLoop { ExternalAccessible := 'False'; ExternalVisible := 'False'; ExternalWritable := 'False'} : Int;
      statEnableRamping { ExternalAccessible := 'False'; ExternalVisible := 'False'; ExternalWritable := 'False'} : Bool;
      statCommandAborted { ExternalAccessible := 'False'; ExternalVisible := 'False'; ExternalWritable := 'False'} : Bool;
      statActualPosition { ExternalAccessible := 'False'; ExternalVisible := 'False'; ExternalWritable := 'False'} : LReal;
      statQOutputForward { ExternalAccessible := 'False'; ExternalVisible := 'False'; ExternalWritable := 'False'} : LReal;
      statQOutputBackward { ExternalAccessible := 'False'; ExternalVisible := 'False'; ExternalWritable := 'False'} : LReal;
      statDirection { ExternalAccessible := 'False'; ExternalVisible := 'False'; ExternalWritable := 'False'} : Byte := #UNDEFINED;
      statMaxPosition { ExternalAccessible := 'False'; ExternalVisible := 'False'; ExternalWritable := 'False'} : LReal;
      statMinPosition { ExternalAccessible := 'False'; ExternalVisible := 'False'; ExternalWritable := 'False'} : LReal;
      statPositionMeasurementStart { ExternalAccessible := 'False'; ExternalVisible := 'False'; ExternalWritable := 'False'} : LReal;
      statPositionMeasurementEnd { ExternalAccessible := 'False'; ExternalVisible := 'False'; ExternalWritable := 'False'} : LReal;
      statActualStepForward { ExternalAccessible := 'False'; ExternalVisible := 'False'; ExternalWritable := 'False'} : Int;
      statActualStepBackward { ExternalAccessible := 'False'; ExternalVisible := 'False'; ExternalWritable := 'False'} : Int;
      statStepCounterMeasurementForwardAborted { ExternalAccessible := 'False'; ExternalVisible := 'False'; ExternalWritable := 'False'} : Int;
      statStepCounterMeasurementBackwardAborted { ExternalAccessible := 'False'; ExternalVisible := 'False'; ExternalWritable := 'False'} : Int;
      statRangeForward { ExternalAccessible := 'False'; ExternalVisible := 'False'; ExternalWritable := 'False'} : Int;
      statRangeBackward { ExternalAccessible := 'False'; ExternalVisible := 'False'; ExternalWritable := 'False'} : Int;
      statIdx { ExternalAccessible := 'False'; ExternalVisible := 'False'; ExternalWritable := 'False'} : Int;
      statActualTime { ExternalAccessible := 'False'; ExternalVisible := 'False'; ExternalWritable := 'False'} : Date_And_Time;
      statTimeMeasurementStart { ExternalAccessible := 'False'; ExternalVisible := 'False'; ExternalWritable := 'False'} : Date_And_Time;
      statTimeMeasurementEnd { ExternalAccessible := 'False'; ExternalVisible := 'False'; ExternalWritable := 'False'} : Date_And_Time;
      statRetInt { ExternalAccessible := 'False'; ExternalVisible := 'False'; ExternalWritable := 'False'} : Int;
      statStatusMeasurement { ExternalAccessible := 'False'; ExternalVisible := 'False'; ExternalWritable := 'False'} : Word;
      statAbortOld { ExternalAccessible := 'False'; ExternalVisible := 'False'; ExternalWritable := 'False'} : Bool;
      statEnableRampingOld { ExternalAccessible := 'False'; ExternalVisible := 'False'; ExternalWritable := 'False'} : Bool;
      statMeasurementForwardDone { ExternalAccessible := 'False'; ExternalVisible := 'False'; ExternalWritable := 'False'} : Bool;
      statMeasurementBackwardDone { ExternalAccessible := 'False'; ExternalVisible := 'False'; ExternalWritable := 'False'} : Bool;
      statConfigForwardOK { ExternalAccessible := 'False'; ExternalVisible := 'False'; ExternalWritable := 'False'} : Bool;
      statConfigBackwardOK { ExternalAccessible := 'False'; ExternalVisible := 'False'; ExternalWritable := 'False'} : Bool;
      instTONWaitForMeasurement {InstructionName := 'TON_TIME'; LibVersion := '1.0'; ExternalAccessible := 'False'; ExternalVisible := 'False'; ExternalWritable := 'False'} : TON_TIME;
      statCoarseBeginBackward { ExternalAccessible := 'False'; ExternalVisible := 'False'; ExternalWritable := 'False'} : Int;
      statCoarseBeginForward { ExternalAccessible := 'False'; ExternalVisible := 'False'; ExternalWritable := 'False'} : Int;
      statForwardFineRangeStepValue { ExternalAccessible := 'False'; ExternalVisible := 'False'; ExternalWritable := 'False'} : Real;
      statForwardCoarseRangeStepValue { ExternalAccessible := 'False'; ExternalVisible := 'False'; ExternalWritable := 'False'} : Real;
      statBackwardFineRangeStepValue { ExternalAccessible := 'False'; ExternalVisible := 'False'; ExternalWritable := 'False'} : Real;
      statBackwardCoarseRangeStepValue { ExternalAccessible := 'False'; ExternalVisible := 'False'; ExternalWritable := 'False'} : Real;
      statEnableRampingMeasurement { ExternalAccessible := 'False'; ExternalVisible := 'False'; ExternalWritable := 'False'} : Bool;
   END_VAR

